KUKA KRL program: MyProgram_295().src

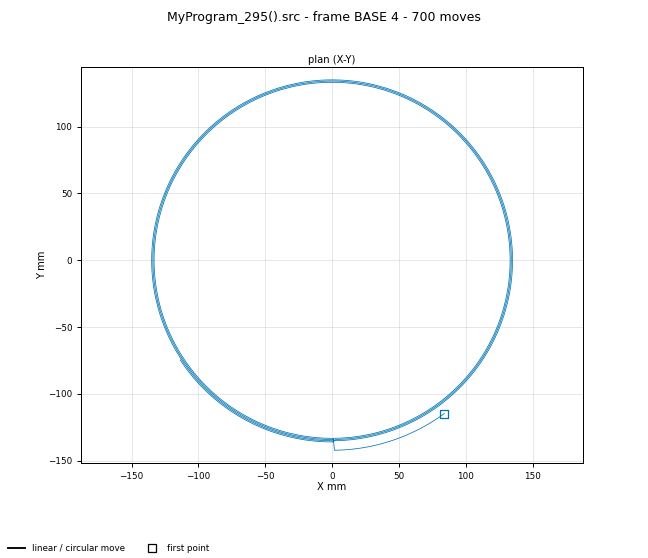
[picture p0: tool path of MyProgram_295().src in frame BASE 4, 700 of 700 moves have a stored position in this frame; points joined in program order, loops and branches not executed]
&ACCESS RVP
&REL 1
&PARAM TEMPLATE = C:\KRC\Roboter\Template\vorgabe
&PARAM EDITMASK = *
DEF MyProgram_295()
; ---- Setting reference (Base) ----
$BASE = BASE_DATA[4]

; --------------------------
; ---- Setting tool (TCP) ----
$TOOL = TOOL_DATA[3]
; --------------------------

$VEL.CP = VEL_APROX_PRINT
Startdeposition()
$VEL.CP = VEL_PRINT
LIN {X 83.9542,Y -114.6488,Z 177,A -50.7197,B 6.574,C 0.3919,E1 6.6804,E2 503.014} C_DIS
LIN {X 80.6167,Y -117.0197,Z 177,A -52.4005,B 6.5737,C 0.3953,E1 6.6765,E2 504.7003} C_DIS
LIN {X 77.4912,Y -119.1123,Z 177,A -53.839,B 6.5737,C 0.3965,E1 6.6732,E2 506.1295} C_DIS
LIN {X 74.5558,Y -120.9716,Z 177,A -55.2209,B 6.5735,C 0.3984,E1 6.6699,E2 507.51} C_DIS
LIN {X 71.534,Y -122.783,Z 177,A -56.6228,B 6.5735,C 0.4003,E1 6.6665,E2 508.9106} C_DIS
LIN {X 68.5439,Y -124.4768,Z 177,A -58.0088,B 6.5733,C 0.4024,E1 6.6632,E2 510.2978} C_DIS
LIN {X 65.0961,Y -126.3132,Z 177,A -59.6809,B 6.573,C 0.4063,E1 6.659,E2 511.9842} C_DIS
LIN {X 61.5313,Y -128.086,Z 177,A -61.1463,B 6.573,C 0.4061,E1 6.6554,E2 513.432} C_DIS
LIN {X 58.3753,Y -129.5551,Z 177,A -62.3689,B 6.5731,C 0.4049,E1 6.6523,E2 514.6314} C_DIS
LIN {X 55.9722,Y -130.6115,Z 177,A -63.5888,B 6.5729,C 0.4089,E1 6.6491,E2 515.8738} C_DIS
LIN {X 52.7667,Y -131.9389,Z 177,A -64.9738,B 6.5728,C 0.4104,E1 6.6456,E2 517.258} C_DIS
LIN {X 49.5072,Y -133.1962,Z 177,A -66.3686,B 6.5728,C 0.4117,E1 6.6419,E2 518.652} C_DIS
LIN {X 46.2416,Y -134.3648,Z 177,A -67.847,B 6.5725,C 0.4145,E1 6.638,E2 520.1421} C_DIS
LIN {X 42.8717,Y -135.4778,Z 177,A -69.1759,B 6.5725,C 0.4143,E1 6.6345,E2 521.4583} C_DIS
LIN {X 39.546,Y -136.4858,Z 177,A -70.5638,B 6.5725,C 0.4154,E1 6.6308,E2 522.8454} C_DIS
LIN {X 36.2237,Y -137.4049,Z 177,A -71.9458,B 6.5725,C 0.4164,E1 6.627,E2 524.2273} C_DIS
LIN {X 32.8538,Y -138.2496,Z 177,A -73.4276,B 6.5723,C 0.4188,E1 6.623,E2 525.7208} C_DIS
LIN {X 29.4326,Y -139.0186,Z 177,A -74.7399,B 6.5723,C 0.4182,E1 6.6194,E2 527.0204} C_DIS
LIN {X 26.0223,Y -139.6976,Z 177,A -76.1321,B 6.5723,C 0.419,E1 6.6156,E2 528.4122} C_DIS
LIN {X 22.581,Y -140.2957,Z 177,A -77.5515,B 6.5722,C 0.42,E1 6.6117,E2 529.834} C_DIS
LIN {X 19.1047,Y -140.8104,Z 177,A -78.9662,B 6.5722,C 0.4207,E1 6.6078,E2 531.2492} C_DIS
LIN {X 15.6477,Y -141.2357,Z 177,A -80.3628,B 6.5722,C 0.4212,E1 6.6039,E2 532.6455} C_DIS
LIN {X 12.1948,Y -141.5751,Z 177,A -81.8408,B 6.572,C 0.423,E1 6.5998,E2 534.1348} C_DIS
LIN {X 8.7227,Y -141.8312,Z 177,A -83.1778,B 6.572,C 0.4224,E1 6.5961,E2 535.4636} C_DIS
LIN {X 5.2085,Y -142.0041,Z 177,A -84.5529,B 6.572,C 0.4221,E1 6.5923,E2 536.8336} C_DIS
LIN {X 1.7271,Y -142.0902,Z 177,A -85.9455,B 6.572,C 0.4221,E1 6.5884,E2 538.2254} C_DIS
LIN {X 1.7271,Y -142.0902,Z 177,A -85.9455,B 6.572,C 0.4221,E1 6.5884,E2 538.2254} C_DIS
Enddeposition()
LIN {X 0.9638,Y -133.1644,Z 178,A -86.3428,B 6.5174,C 0.3854,E1 6.5313,E2 538.3182} C_DIS
Startdeposition()
$VEL.CP = VEL_PRINT
LIN {X 4.5117,Y -133.0931,Z 178,A -84.4,B 6.5178,C 0.3791,E1 6.5369,E2 536.3228} C_DIS
LIN {X 7.0319,Y -132.9825,Z 178,A -83.1818,B 6.5179,C 0.3769,E1 6.5404,E2 535.0873} C_DIS
LIN {X 10.9069,Y -132.7207,Z 178,A -81.6183,B 6.5179,C 0.3779,E1 6.5447,E2 533.5364} C_DIS
LIN {X 13.8082,Y -132.4506,Z 178,A -80.2868,B 6.5179,C 0.3763,E1 6.5484,E2 532.1945} C_DIS
LIN {X 17.4081,Y -132.025,Z 178,A -78.8233,B 6.5179,C 0.3769,E1 6.5524,E2 530.7422} C_DIS
LIN {X 21.1427,Y -131.4808,Z 178,A -77.1933,B 6.5179,C 0.3759,E1 6.5569,E2 529.1105} C_DIS
LIN {X 24.3569,Y -130.9228,Z 178,A -75.7994,B 6.518,C 0.3752,E1 6.5608,E2 527.7169} C_DIS
LIN {X 27.3232,Y -130.3367,Z 178,A -74.425,B 6.5182,C 0.3732,E1 6.5646,E2 526.3324} C_DIS
LIN {X 30.7671,Y -129.5653,Z 178,A -72.8889,B 6.5182,C 0.3718,E1 6.5687,E2 524.7932} C_DIS
LIN {X 35.009,Y -128.4853,Z 178,A -70.9984,B 6.5183,C 0.3701,E1 6.5739,E2 522.9005} C_DIS
LIN {X 39.1367,Y -127.2867,Z 178,A -69.2948,B 6.5183,C 0.3706,E1 6.5784,E2 521.2139} C_DIS
LIN {X 42.8597,Y -126.0843,Z 178,A -67.6307,B 6.5183,C 0.3692,E1 6.5828,E2 519.5511} C_DIS
LIN {X 46.8767,Y -124.6441,Z 178,A -65.7393,B 6.5185,C 0.3663,E1 6.5878,E2 517.6514} C_DIS
LIN {X 50.4594,Y -123.2392,Z 178,A -64.161,B 6.5185,C 0.3656,E1 6.5918,E2 516.0816} C_DIS
LIN {X 53.9636,Y -121.7442,Z 178,A -62.5457,B 6.5187,C 0.3639,E1 6.596,E2 514.468} C_DIS
LIN {X 56.9303,Y -120.3858,Z 178,A -61.1578,B 6.5187,C 0.3623,E1 6.5995,E2 513.0811} C_DIS
LIN {X 59.8618,Y -118.9557,Z 178,A -59.7718,B 6.5189,C 0.3606,E1 6.6029,E2 511.6962} C_DIS
LIN {X 62.7544,Y -117.4566,Z 178,A -58.3828,B 6.5189,C 0.3588,E1 6.6064,E2 510.3076} C_DIS
LIN {X 65.6366,Y -115.8708,Z 178,A -56.9757,B 6.5191,C 0.3568,E1 6.6098,E2 508.9005} C_DIS
LIN {X 68.0271,Y -114.4832,Z 178,A -55.71,B 6.5192,C 0.3538,E1 6.6129,E2 507.6242} C_DIS
LIN {X 71.6806,Y -112.2317,Z 178,A -53.8771,B 6.5194,C 0.351,E1 6.6172,E2 505.7914} C_DIS
LIN {X 74.9099,Y -110.103,Z 178,A -52.4203,B 6.5194,C 0.3515,E1 6.6205,E2 504.3592} C_DIS
LIN {X 77.5879,Y -108.2321,Z 178,A -50.9492,B 6.5195,C 0.348,E1 6.6239,E2 502.8786} C_DIS
LIN {X 80.6412,Y -105.9771,Z 178,A -49.228,B 6.5198,C 0.3437,E1 6.6278,E2 501.1451} C_DIS
LIN {X 83.8487,Y -103.4579,Z 178,A -47.5664,B 6.5198,C 0.3419,E1 6.6314,E2 499.4936} C_DIS
LIN {X 86.7837,Y -101.0083,Z 178,A -45.8978,B 6.52,C 0.3383,E1 6.635,E2 497.8205} C_DIS
LIN {X 90.026,Y -98.1295,Z 178,A -44.057,B 6.5202,C 0.335,E1 6.6388,E2 495.9812} C_DIS
LIN {X 93.0048,Y -95.3115,Z 178,A -42.3038,B 6.5204,C 0.3315,E1 6.6423,E2 494.2277} C_DIS
LIN {X 95.8799,Y -92.4185,Z 178,A -40.5795,B 6.5206,C 0.3283,E1 6.6457,E2 492.5057} C_DIS
LIN {X 98.8364,Y -89.2498,Z 178,A -38.744,B 6.5207,C 0.3247,E1 6.6491,E2 490.6721} C_DIS
LIN {X 101.7336,Y -85.9331,Z 178,A -36.8835,B 6.5209,C 0.3211,E1 6.6525,E2 488.8141} C_DIS
LIN {X 104.4775,Y -82.5752,Z 178,A -35.0437,B 6.5211,C 0.3172,E1 6.6557,E2 486.9759} C_DIS
LIN {X 106.9568,Y -79.337,Z 178,A -33.4349,B 6.5211,C 0.3156,E1 6.6584,E2 485.3836} C_DIS
LIN {X 108.8683,Y -76.6925,Z 178,A -32.0564,B 6.5213,C 0.3126,E1 6.6606,E2 484.007} C_DIS
LIN {X 111.0112,Y -73.5576,Z 178,A -30.3322,B 6.5216,C 0.3071,E1 6.6633,E2 482.2701} C_DIS
LIN {X 113.0997,Y -70.303,Z 178,A -28.7379,B 6.5217,C 0.3042,E1 6.6657,E2 480.6828} C_DIS
LIN {X 115.0507,Y -67.0639,Z 178,A -27.1021,B 6.5219,C 0.3,E1 6.668,E2 479.0444} C_DIS
LIN {X 117.2134,Y -63.207,Z 178,A -25.2998,B 6.5221,C 0.2968,E1 6.6704,E2 477.2528} C_DIS
LIN {X 118.7218,Y -60.3213,Z 178,A -23.9903,B 6.5221,C 0.2947,E1 6.6721,E2 475.9532} C_DIS
LIN {X 120.1639,Y -57.3948,Z 178,A -22.6669,B 6.5223,C 0.2924,E1 6.6737,E2 474.6386} C_DIS
LIN {X 121.5341,Y -54.4334,Z 178,A -21.1584,B 6.5225,C 0.2869,E1 6.6754,E2 473.1158} C_DIS
LIN {X 123.0296,Y -50.9648,Z 178,A -19.5935,B 6.5226,C 0.2836,E1 6.6771,E2 471.5568} C_DIS
LIN {X 124.6437,Y -46.8779,Z 178,A -17.7069,B 6.5229,C 0.2786,E1 6.679,E2 469.669} C_DIS
LIN {X 125.9218,Y -43.3284,Z 178,A -16.2072,B 6.5229,C 0.2762,E1 6.6804,E2 468.1831} C_DIS
LIN {X 126.9445,Y -40.2337,Z 178,A -14.8581,B 6.5231,C 0.2733,E1 6.6816,E2 466.8393} C_DIS
LIN {X 127.8843,Y -37.1383,Z 178,A -13.4781,B 6.5232,C 0.2696,E1 6.6827,E2 465.4595} C_DIS
LIN {X 128.7261,Y -34.1058,Z 178,A -12.1735,B 6.5234,C 0.2667,E1 6.6836,E2 464.1598} C_DIS
LIN {X 129.6834,Y -30.2687,Z 178,A -10.3349,B 6.5236,C 0.2596,E1 6.6848,E2 462.3028} C_DIS
LIN {X 130.5066,Y -26.4881,Z 178,A -8.8533,B 6.5237,C 0.258,E1 6.6857,E2 460.8423} C_DIS
LIN {X 131.1169,Y -23.281,Z 178,A -7.4791,B 6.5238,C 0.2546,E1 6.6864,E2 459.4707} C_DIS
LIN {X 131.6511,Y -20.0427,Z 178,A -6.0255,B 6.524,C 0.2499,E1 6.687,E2 458.0106} C_DIS
LIN {X 132.1671,Y -16.3023,Z 178,A -4.4968,B 6.5241,C 0.2469,E1 6.6875,E2 456.4924} C_DIS
LIN {X 132.5264,Y -13.0578,Z 178,A -3.1273,B 6.5243,C 0.2435,E1 6.6879,E2 455.126} C_DIS
LIN {X 132.8063,Y -9.8053,Z 178,A -1.7588,B 6.5243,C 0.2401,E1 6.6882,E2 453.7608} C_DIS
LIN {X 133.0068,Y -6.547,Z 178,A -0.3905,B 6.5245,C 0.2366,E1 6.6884,E2 452.3957} C_DIS
LIN {X 133.1405,Y -2.7529,Z 178,A 1.3295,B 6.5247,C 0.2305,E1 6.6886,E2 450.6637} C_DIS
LIN {X 133.1592,Y 1.6279,Z 178,A 3.1809,B 6.5249,C 0.2257,E1 6.6886,E2 448.8149} C_DIS
LIN {X 133.0343,Y 6.0011,Z 178,A 4.8481,B 6.5249,C 0.2239,E1 6.6884,E2 447.1727} C_DIS
LIN {X 132.8441,Y 9.2877,Z 178,A 6.2915,B 6.5251,C 0.2194,E1 6.6881,E2 445.7248} C_DIS
LIN {X 132.5762,Y 12.5389,Z 178,A 7.6588,B 6.5252,C 0.2161,E1 6.6878,E2 444.3609} C_DIS
LIN {X 132.2291,Y 15.7828,Z 178,A 9.0275,B 6.5253,C 0.2127,E1 6.6874,E2 442.9954} C_DIS
LIN {X 131.803,Y 19.0166,Z 178,A 10.4532,B 6.5255,C 0.2083,E1 6.6868,E2 441.566} C_DIS
LIN {X 131.2089,Y 22.7666,Z 178,A 11.9579,B 6.5255,C 0.2059,E1 6.6861,E2 440.0759} C_DIS
LIN {X 130.6108,Y 25.976,Z 178,A 13.5008,B 6.5257,C 0.1996,E1 6.6853,E2 438.5151} C_DIS
LIN {X 129.686,Y 30.2575,Z 178,A 15.1757,B 6.5257,C 0.1979,E1 6.6843,E2 436.8646} C_DIS
LIN {X 129.0503,Y 32.8574,Z 178,A 16.4149,B 6.5259,C 0.1932,E1 6.6834,E2 435.6138} C_DIS
LIN {X 128.0423,Y 36.5967,Z 178,A 17.964,B 6.526,C 0.1906,E1 6.6823,E2 434.078} C_DIS
LIN {X 127.1068,Y 39.7246,Z 178,A 19.3402,B 6.5261,C 0.1873,E1 6.6812,E2 432.7044} C_DIS
LIN {X 125.5625,Y 44.3647,Z 178,A 21.6447,B 6.5264,C 0.1782,E1 6.6791,E2 430.3742} C_DIS
LIN {X 123.8678,Y 48.8956,Z 178,A 23.4542,B 6.5264,C 0.1772,E1 6.6773,E2 428.5966} C_DIS
LIN {X 122.6601,Y 51.8494,Z 178,A 24.934,B 6.5265,C 0.1718,E1 6.6757,E2 427.1029} C_DIS
LIN {X 121.0791,Y 55.4403,Z 178,A 26.4508,B 6.5265,C 0.1703,E1 6.674,E2 425.606} C_DIS
LIN {X 119.678,Y 58.404,Z 178,A 27.8275,B 6.5266,C 0.1672,E1 6.6723,E2 424.2328} C_DIS
LIN {X 118.4793,Y 60.7976,Z 178,A 28.9716,B 6.5267,C 0.1644,E1 6.6709,E2 423.089} C_DIS
LIN {X 116.8622,Y 63.8538,Z 178,A 30.4879,B 6.5268,C 0.1602,E1 6.6688,E2 421.5685} C_DIS
LIN {X 115.0507,Y 67.0638,Z 178,A 31.9027,B 6.5268,C 0.1591,E1 6.6669,E2 420.1737} C_DIS
LIN {X 113.3731,Y 69.8617,Z 178,A 33.4559,B 6.527,C 0.1532,E1 6.6646,E2 418.6017} C_DIS
LIN {X 111.0211,Y 73.5425,Z 178,A 35.2069,B 6.527,C 0.1508,E1 6.662,E2 416.8655} C_DIS
LIN {X 109.1792,Y 76.2497,Z 178,A 36.5869,B 6.5271,C 0.148,E1 6.6598,E2 415.4883} C_DIS
LIN {X 107.2785,Y 78.9011,Z 178,A 37.925,B 6.5271,C 0.1458,E1 6.6576,E2 414.1576} C_DIS
LIN {X 105.0146,Y 81.891,Z 178,A 39.591,B 6.5273,C 0.1413,E1 6.6548,E2 412.4848} C_DIS
LIN {X 102.5253,Y 84.9859,Z 178,A 41.3184,B 6.5273,C 0.1372,E1 6.6517,E2 410.7545} C_DIS
LIN {X 99.5928,Y 88.4047,Z 178,A 43.2432,B 6.5274,C 0.1332,E1 6.6482,E2 408.8307} C_DIS
LIN {X 96.6295,Y 91.6347,Z 178,A 45.0403,B 6.5274,C 0.1307,E1 6.6448,E2 407.0439} C_DIS
LIN {X 93.806,Y 94.5224,Z 178,A 46.749,B 6.5275,C 0.1276,E1 6.6414,E2 405.3381} C_DIS
LIN {X 90.8317,Y 97.3841,Z 178,A 48.5361,B 6.5276,C 0.124,E1 6.6378,E2 403.5493} C_DIS
LIN {X 87.6175,Y 100.2858,Z 178,A 50.3796,B 6.5276,C 0.1207,E1 6.6339,E2 401.7077} C_DIS
LIN {X 84.2856,Y 103.1018,Z 178,A 52.2249,B 6.5277,C 0.1178,E1 6.63,E2 399.866} C_DIS
LIN {X 80.847,Y 105.8198,Z 178,A 54.0372,B 6.5277,C 0.1156,E1 6.626,E2 398.0623} C_DIS
LIN {X 78.3357,Y 107.6923,Z 178,A 55.396,B 6.5278,C 0.1132,E1 6.623,E2 396.702} C_DIS
LIN {X 75.4138,Y 109.758,Z 178,A 56.8258,B 6.5278,C 0.1123,E1 6.6197,E2 395.2852} C_DIS
LIN {X 72.8869,Y 111.4528,Z 178,A 58.1198,B 6.5278,C 0.1105,E1 6.6167,E2 393.993} C_DIS
LIN {X 70.3001,Y 113.1016,Z 178,A 59.529,B 6.5279,C 0.1071,E1 6.6133,E2 392.573} C_DIS
LIN {X 67.0645,Y 115.0503,Z 178,A 60.9746,B 6.5279,C 0.1074,E1 6.6099,E2 391.1489} C_DIS
LIN {X 64.6771,Y 116.4087,Z 178,A 62.2133,B 6.5279,C 0.1049,E1 6.6069,E2 389.9033} C_DIS
LIN {X 61.8012,Y 117.9582,Z 178,A 63.6121,B 6.5279,C 0.1031,E1 6.6034,E2 388.5053} C_DIS
LIN {X 58.8644,Y 119.4508,Z 178,A 65.0105,B 6.5279,C 0.1016,E1 6.5999,E2 387.1092} C_DIS
LIN {X 55.9201,Y 120.8572,Z 178,A 66.4007,B 6.528,C 0.1,E1 6.5964,E2 385.7207} C_DIS
LIN {X 52.4684,Y 122.396,Z 178,A 68.0149,B 6.528,C 0.0983,E1 6.5923,E2 384.1081} C_DIS
LIN {X 48.9807,Y 123.8348,Z 178,A 69.7866,B 6.5281,C 0.0944,E1 6.5877,E2 382.3189} C_DIS
LIN {X 44.8735,Y 125.3795,Z 178,A 71.4956,B 6.5281,C 0.0951,E1 6.5833,E2 380.6315} C_DIS
LIN {X 41.772,Y 126.4467,Z 178,A 72.8947,B 6.5281,C 0.094,E1 6.5796,E2 379.2341} C_DIS
LIN {X 38.6838,Y 127.4253,Z 178,A 74.2776,B 6.5281,C 0.093,E1 6.5759,E2 377.8527} C_DIS
LIN {X 35.5863,Y 128.3249,Z 178,A 75.6541,B 6.5281,C 0.092,E1 6.5722,E2 376.4779} C_DIS
LIN {X 32.5276,Y 129.134,Z 178,A 77.1152,B 6.5281,C 0.0896,E1 6.5682,E2 375.0052} C_DIS
LIN {X 28.0899,Y 130.1713,Z 178,A 78.9048,B 6.5281,C 0.0908,E1 6.5634,E2 373.2365} C_DIS
LIN {X 24.8792,Y 130.823,Z 178,A 80.3656,B 6.5281,C 0.0892,E1 6.5593,E2 371.77} C_DIS
LIN {X 21.6641,Y 131.3939,Z 178,A 81.7621,B 6.5281,C 0.0887,E1 6.5555,E2 370.3749} C_DIS
LIN {X 18.5251,Y 131.8732,Z 178,A 83.227,B 6.5282,C 0.0867,E1 6.5514,E2 368.8987} C_DIS
LIN {X 14.6874,Y 132.356,Z 178,A 84.7973,B 6.5282,C 0.0874,E1 6.5471,E2 367.3402} C_DIS
LIN {X 11.4395,Y 132.6757,Z 178,A 86.1979,B 6.5282,C 0.0871,E1 6.5432,E2 365.9406} C_DIS
LIN {X 8.1676,Y 132.9171,Z 178,A 87.6578,B 6.5282,C 0.0861,E1 6.5391,E2 364.4754} C_DIS
LIN {X 3.7923,Y 133.1139,Z 178,A 89.552,B 6.5282,C 0.0857,E1 6.5338,E2 362.5808} C_DIS
LIN {X 0.018,Y 133.1698,Z 178,A 91.0729,B 6.5282,C 0.0871,E1 6.5296,E2 361.073} C_DIS
LIN {X -2.7571,Y 133.1404,Z 178,A 92.4181,B 6.5282,C 0.0851,E1 6.5258,E2 359.7104} C_DIS
LIN {X -6.5309,Y 133.0076,Z 178,A 94.0135,B 6.5282,C 0.0857,E1 6.5214,E2 358.1192} C_DIS
LIN {X -10.9,Y 132.7213,Z 178,A 95.8193,B 6.5282,C 0.0871,E1 6.5164,E2 356.3236} C_DIS
LIN {X -14.16,Y 132.4128,Z 178,A 97.2257,B 6.5282,C 0.0875,E1 6.5125,E2 354.9182} C_DIS
LIN {X -17.4113,Y 132.0246,Z 178,A 98.6351,B 6.5282,C 0.0879,E1 6.5086,E2 353.5095} C_DIS
LIN {X -21.1485,Y 131.4799,Z 178,A 100.2795,B 6.5282,C 0.0884,E1 6.504,E2 351.8638} C_DIS
LIN {X -24.3644,Y 130.9214,Z 178,A 101.6857,B 6.5282,C 0.089,E1 6.5002,E2 350.4582} C_DIS
LIN {X -27.5659,Y 130.2844,Z 178,A 103.0938,B 6.5282,C 0.0898,E1 6.4963,E2 349.0505} C_DIS
LIN {X -30.7693,Y 129.5648,Z 178,A 104.6246,B 6.5282,C 0.0891,E1 6.4921,E2 347.5065} C_DIS
LIN {X -35.0164,Y 128.4833,Z 178,A 106.4004,B 6.5282,C 0.0919,E1 6.4874,E2 345.7449} C_DIS
LIN {X -37.5751,Y 127.7564,Z 178,A 107.6249,B 6.5282,C 0.0918,E1 6.484,E2 344.5116} C_DIS
LIN {X -40.7134,Y 126.7912,Z 178,A 109.0414,B 6.5282,C 0.0929,E1 6.4803,E2 343.0956} C_DIS
LIN {X -44.3614,Y 125.5637,Z 178,A 110.8869,B 6.5282,C 0.0921,E1 6.4753,E2 341.2288} C_DIS
LIN {X -48.9142,Y 123.8606,Z 178,A 112.7575,B 6.5281,C 0.097,E1 6.4705,E2 339.3859} C_DIS
LIN {X -51.9858,Y 122.6031,Z 178,A 114.3234,B 6.5281,C 0.0968,E1 6.4665,E2 337.8046} C_DIS
LIN {X -55.4531,Y 121.0732,Z 178,A 115.8357,B 6.5281,C 0.1002,E1 6.4627,E2 336.3076} C_DIS
LIN {X -58.4045,Y 119.6777,Z 178,A 117.1617,B 6.528,C 0.1028,E1 6.4593,E2 334.992} C_DIS
LIN {X -61.3202,Y 118.2108,Z 178,A 118.6541,B 6.528,C 0.1036,E1 6.4556,E2 333.4902} C_DIS
LIN {X -63.7257,Y 116.932,Z 178,A 119.9582,B 6.528,C 0.1036,E1 6.4524,E2 332.1713} C_DIS
LIN {X -66.7643,Y 115.2241,Z 178,A 121.3384,B 6.528,C 0.1071,E1 6.4491,E2 330.8065} C_DIS
LIN {X -69.4067,Y 113.6523,Z 178,A 122.82,B 6.528,C 0.1071,E1 6.4455,E2 329.3071} C_DIS
LIN {X -72.8951,Y 111.4474,Z 178,A 124.6638,B 6.5279,C 0.1091,E1 6.4411,E2 327.4566} C_DIS
LIN {X -76.1879,Y 109.2222,Z 178,A 126.2443,B 6.5279,C 0.1134,E1 6.4375,E2 325.8929} C_DIS
LIN {X -78.9118,Y 107.2706,Z 178,A 127.8007,B 6.5278,C 0.1145,E1 6.434,E2 324.324} C_DIS
LIN {X -82.3732,Y 104.6362,Z 178,A 129.6469,B 6.5278,C 0.1181,E1 6.4299,E2 322.4824} C_DIS
LIN {X -85.3094,Y 102.2571,Z 178,A 131.3251,B 6.5277,C 0.1204,E1 6.4263,E2 320.7994} C_DIS
LIN {X -88.4026,Y 99.5947,Z 178,A 133.1508,B 6.5277,C 0.1229,E1 6.4224,E2 318.9669} C_DIS
LIN {X -91.4919,Y 96.7641,Z 178,A 134.9499,B 6.5276,C 0.1265,E1 6.4188,E2 317.1698} C_DIS
LIN {X -94.5601,Y 93.7681,Z 178,A 136.7855,B 6.5275,C 0.1303,E1 6.4151,E2 315.3369} C_DIS
LIN {X -97.3895,Y 90.8259,Z 178,A 138.6197,B 6.5275,C 0.1331,E1 6.4116,E2 313.495} C_DIS
LIN {X -100.2963,Y 87.6054,Z 178,A 140.5235,B 6.5274,C 0.1366,E1 6.4081,E2 311.5884} C_DIS
LIN {X -103.1045,Y 84.2824,Z 178,A 142.4264,B 6.5273,C 0.1404,E1 6.4047,E2 309.6836} C_DIS
LIN {X -105.8227,Y 80.8432,Z 178,A 144.2965,B 6.5272,C 0.1449,E1 6.4015,E2 307.8171} C_DIS
LIN {X -107.9243,Y 78.0156,Z 178,A 145.7984,B 6.5271,C 0.1485,E1 6.399,E2 306.3182} C_DIS
LIN {X -109.811,Y 75.3366,Z 178,A 147.3294,B 6.5271,C 0.1505,E1 6.3965,E2 304.774} C_DIS
LIN {X -112.2487,Y 71.6541,Z 178,A 149.1704,B 6.5269,C 0.1558,E1 6.3937,E2 302.9418} C_DIS
LIN {X -114.2296,Y 68.4525,Z 178,A 150.8148,B 6.5269,C 0.1595,E1 6.3913,E2 301.296} C_DIS
LIN {X -115.6178,Y 66.0802,Z 178,A 152.0242,B 6.5268,C 0.1621,E1 6.3896,E2 300.0844} C_DIS
LIN {X -117.1999,Y 63.2321,Z 178,A 153.5274,B 6.5268,C 0.1645,E1 6.3876,E2 298.5704} C_DIS
LIN {X -118.7111,Y 60.3422,Z 178,A 155.0025,B 6.5266,C 0.1673,E1 6.3857,E2 297.0879} C_DIS
LIN {X -120.7967,Y 56.051,Z 178,A 157.0993,B 6.5266,C 0.1722,E1 6.3832,E2 294.9877} C_DIS
LIN {X -122.3961,Y 52.468,Z 178,A 158.7111,B 6.5264,C 0.1774,E1 6.3814,E2 293.3866} C_DIS
LIN {X -123.84,Y 48.9671,Z 178,A 160.5404,B 6.5264,C 0.1796,E1 6.3795,E2 291.5349} C_DIS
LIN {X -125.3863,Y 44.8545,Z 178,A 162.3044,B 6.5261,C 0.1861,E1 6.3778,E2 289.7877} C_DIS
LIN {X -126.4476,Y 41.769,Z 178,A 163.7384,B 6.5261,C 0.1896,E1 6.3765,E2 288.3514} C_DIS
LIN {X -127.4332,Y 38.6583,Z 178,A 165.1722,B 6.5259,C 0.1931,E1 6.3753,E2 286.9152} C_DIS
LIN {X -128.3421,Y 35.5246,Z 178,A 166.6066,B 6.5259,C 0.1967,E1 6.3743,E2 285.4785} C_DIS
LIN {X -129.1739,Y 32.3705,Z 178,A 168.1162,B 6.5257,C 0.1994,E1 6.3732,E2 283.9574} C_DIS
LIN {X -130.1662,Y 28.1131,Z 178,A 169.8859,B 6.5255,C 0.2059,E1 6.3721,E2 282.2027} C_DIS
LIN {X -130.824,Y 24.8739,Z 178,A 171.4189,B 6.5255,C 0.2087,E1 6.3713,E2 280.6576} C_DIS
LIN {X -131.3947,Y 21.6592,Z 178,A 172.8531,B 6.5253,C 0.2124,E1 6.3706,E2 279.2211} C_DIS
LIN {X -131.9575,Y 17.923,Z 178,A 174.6577,B 6.5253,C 0.2151,E1 6.3699,E2 277.3963} C_DIS
LIN {X -132.4646,Y 13.6779,Z 178,A 176.5493,B 6.5251,C 0.2198,E1 6.3693,E2 275.5} C_DIS
LIN {X -132.8073,Y 9.7921,Z 178,A 178.1203,B 6.5249,C 0.2257,E1 6.369,E2 273.9433} C_DIS
LIN {X -133.0334,Y 6.0183,Z 178,A 179.9405,B 6.5249,C 0.2283,E1 6.3687,E2 272.1011} C_DIS
LIN {X -133.159,Y 1.6377,Z 178,A -178.3452,B 6.5245,C 0.2355,E1 6.3686,E2 270.4091} C_DIS
LIN {X -133.1592,Y -1.6294,Z 178,A -176.7176,B 6.5245,C 0.2372,E1 6.3686,E2 268.7557} C_DIS
LIN {X -133.0332,Y -6.0233,Z 178,A -174.9739,B 6.5242,C 0.2442,E1 6.3688,E2 267.0314} C_DIS
LIN {X -132.8445,Y -9.2821,Z 178,A -173.4663,B 6.5242,C 0.2471,E1 6.3691,E2 265.5123} C_DIS
LIN {X -132.5763,Y -12.5379,Z 178,A -172.0358,B 6.524,C 0.2508,E1 6.3694,E2 264.0799} C_DIS
LIN {X -132.2289,Y -15.7845,Z 178,A -170.6013,B 6.5238,C 0.2545,E1 6.3699,E2 262.6428} C_DIS
LIN {X -131.8007,Y -19.0321,Z 178,A -169.1108,B 6.5238,C 0.2576,E1 6.3704,E2 261.1434} C_DIS
LIN {X -131.2089,Y -22.7668,Z 178,A -167.4875,B 6.5235,C 0.2622,E1 6.3712,E2 259.5218} C_DIS
LIN {X -130.6106,Y -25.9774,Z 178,A -166.054,B 6.5234,C 0.2658,E1 6.372,E2 258.0859} C_DIS
LIN {X -129.9358,Y -29.1637,Z 178,A -164.5219,B 6.5233,C 0.2683,E1 6.3729,E2 256.5387} C_DIS
LIN {X -128.9703,Y -33.1725,Z 178,A -162.8528,B 6.523,C 0.2744,E1 6.374,E2 254.8837} C_DIS
LIN {X -128.0384,Y -36.6106,Z 178,A -161.2582,B 6.5229,C 0.2779,E1 6.3752,E2 253.2826} C_DIS
LIN {X -127.1124,Y -39.7064,Z 178,A -159.8377,B 6.5227,C 0.2813,E1 6.3764,E2 251.8593} C_DIS
LIN {X -126.0941,Y -42.8309,Z 178,A -158.3821,B 6.5226,C 0.2847,E1 6.3776,E2 250.3995} C_DIS
LIN {X -124.6478,Y -46.8667,Z 178,A -156.4284,B 6.5224,C 0.2884,E1 6.3795,E2 248.4335} C_DIS
LIN {X -123.4191,Y -50.0133,Z 178,A -154.9576,B 6.5223,C 0.292,E1 6.3811,E2 246.9614} C_DIS
LIN {X -121.8155,Y -53.8043,Z 178,A -153.1555,B 6.5221,C 0.2963,E1 6.3831,E2 245.1565} C_DIS
LIN {X -120.3852,Y -56.9316,Z 178,A -151.8109,B 6.5218,C 0.3016,E1 6.3846,E2 243.8292} C_DIS
LIN {X -119.0565,Y -59.6637,Z 178,A -150.3536,B 6.5218,C 0.3032,E1 6.3864,E2 242.3543} C_DIS
LIN {X -117.4544,Y -62.7585,Z 178,A -148.8411,B 6.5216,C 0.3068,E1 6.3884,E2 240.8409} C_DIS
LIN {X -115.6453,Y -66.0319,Z 178,A -147.0877,B 6.5215,C 0.3091,E1 6.3908,E2 239.0705} C_DIS
LIN {X -113.3745,Y -69.8595,Z 178,A -145.1363,B 6.5213,C 0.3133,E1 6.3937,E2 237.1155} C_DIS
LIN {X -111.0145,Y -73.5526,Z 178,A -143.2028,B 6.5211,C 0.3172,E1 6.3966,E2 235.1769} C_DIS
LIN {X -108.5248,Y -77.1786,Z 178,A -141.2843,B 6.5209,C 0.3212,E1 6.3997,E2 233.2559} C_DIS
LIN {X -105.9892,Y -80.6255,Z 178,A -139.4011,B 6.5207,C 0.3249,E1 6.4028,E2 231.3683} C_DIS
LIN {X -103.4756,Y -83.8268,Z 178,A -137.6864,B 6.5205,C 0.3291,E1 6.4058,E2 229.6587} C_DIS
LIN {X -101.0063,Y -86.786,Z 178,A -135.9543,B 6.5204,C 0.3317,E1 6.409,E2 227.9179} C_DIS
LIN {X -98.1174,Y -90.0391,Z 178,A -134.0489,B 6.5202,C 0.3352,E1 6.4125,E2 226.0089} C_DIS
LIN {X -95.3144,Y -93.0018,Z 178,A -132.2472,B 6.5201,C 0.3381,E1 6.416,E2 224.2019} C_DIS
LIN {X -92.4219,Y -95.8766,Z 178,A -130.4685,B 6.5199,C 0.3412,E1 6.4196,E2 222.4206} C_DIS
LIN {X -89.4427,Y -98.6613,Z 178,A -128.699,B 6.5197,C 0.3443,E1 6.4232,E2 220.6497} C_DIS
LIN {X -86.3647,Y -101.3668,Z 178,A -126.962,B 6.5196,C 0.3478,E1 6.4269,E2 218.9162} C_DIS
LIN {X -83.2179,Y -103.9662,Z 178,A -125.1123,B 6.5195,C 0.3497,E1 6.4309,E2 217.0551} C_DIS
LIN {X -79.8155,Y -106.6005,Z 178,A -123.2351,B 6.5193,C 0.3524,E1 6.4351,E2 215.1749} C_DIS
LIN {X -76.7046,Y -108.8599,Z 178,A -121.7,B 6.5191,C 0.3565,E1 6.4386,E2 213.6548} C_DIS
LIN {X -73.5588,Y -111.0104,Z 178,A -119.8949,B 6.5191,C 0.3569,E1 6.4428,E2 211.8293} C_DIS
LIN {X -70.3041,Y -113.099,Z 178,A -118.2513,B 6.5189,C 0.3595,E1 6.4467,E2 210.1883} C_DIS
LIN {X -67.0675,Y -115.0486,Z 178,A -116.7722,B 6.5187,C 0.3636,E1 6.4502,E2 208.7274} C_DIS
LIN {X -64.8802,Y -116.2962,Z 178,A -115.6142,B 6.5187,C 0.3641,E1 6.453,E2 207.5602} C_DIS
LIN {X -61.779,Y -117.9699,Z 178,A -114.0708,B 6.5186,C 0.3656,E1 6.4568,E2 206.0132} C_DIS
LIN {X -58.8692,Y -119.4485,Z 178,A -112.6543,B 6.5185,C 0.3671,E1 6.4604,E2 204.5951} C_DIS
LIN {X -55.924,Y -120.8554,Z 178,A -111.2464,B 6.5185,C 0.3686,E1 6.4639,E2 203.1867} C_DIS
LIN {X -52.4719,Y -122.3944,Z 178,A -109.5959,B 6.5183,C 0.37,E1 6.4682,E2 201.533} C_DIS
LIN {X -48.9846,Y -123.8332,Z 178,A -107.7957,B 6.5183,C 0.3693,E1 6.4729,E2 199.7106} C_DIS
LIN {X -44.8617,Y -125.3837,Z 178,A -106.0552,B 6.5182,C 0.3729,E1 6.4774,E2 197.9891} C_DIS
LIN {X -41.7968,Y -126.4384,Z 178,A -104.6531,B 6.5182,C 0.374,E1 6.4811,E2 196.5857} C_DIS
LIN {X -38.7182,Y -127.4148,Z 178,A -103.2584,B 6.5181,C 0.3749,E1 6.4848,E2 195.1901} C_DIS
LIN {X -35.6645,Y -128.303,Z 178,A -101.8975,B 6.518,C 0.3759,E1 6.4885,E2 193.8299} C_DIS
LIN {X -32.3623,Y -129.176,Z 178,A -100.3256,B 6.518,C 0.3754,E1 6.4928,E2 192.2448} C_DIS
LIN {X -28.0815,Y -130.173,Z 178,A -98.5028,B 6.518,C 0.3773,E1 6.4977,E2 190.43} C_DIS
LIN {X -25.1996,Y -130.7617,Z 178,A -97.1703,B 6.518,C 0.377,E1 6.5014,E2 189.0888} C_DIS
LIN {X -21.6685,Y -131.3931,Z 178,A -95.6898,B 6.5179,C 0.3784,E1 6.5055,E2 187.6156} C_DIS
LIN {X -17.9346,Y -131.956,Z 178,A -94.0441,B 6.5179,C 0.3786,E1 6.51,E2 185.9667} C_DIS
LIN {X -14.6925,Y -132.3555,Z 178,A -92.6346,B 6.5179,C 0.3788,E1 6.5139,E2 184.5562} C_DIS
LIN {X -11.427,Y -132.6767,Z 178,A -91.2309,B 6.5179,C 0.3791,E1 6.5178,E2 183.1529} C_DIS
LIN {X -8.1726,Y -132.9168,Z 178,A -89.7714,B 6.5179,C 0.3784,E1 6.5219,E2 181.6859} C_DIS
LIN {X -3.8022,Y -133.1136,Z 178,A -87.8767,B 6.5179,C 0.3782,E1 6.5272,E2 179.7889} C_DIS
LIN {X -0.0979,Y -133.1694,Z 178,A -86.3929,B 6.5178,C 0.3797,E1 6.5313,E2 178.3182} C_DIS
LIN {X -0.0979,Y -133.1694,Z 178,A -86.3929,B 6.5178,C 0.3797,E1 6.5313,E2 178.3182} C_DIS
Enddeposition()
LIN {X 0.9658,Y -134.0683,Z 178,A -86.4358,B 6.517,C 0.3905,E1 6.5308,E2 178.4564} C_DIS
Startdeposition()
$VEL.CP = VEL_PRINT
LIN {X -2.4569,Y -134.0498,Z 178,A -88.0612,B 6.5169,C 0.3929,E1 6.5262,E2 180.1028} C_DIS
LIN {X -6.2008,Y -133.9296,Z 178,A -89.7044,B 6.5169,C 0.3935,E1 6.5216,E2 181.752} C_DIS
LIN {X -10.5469,Y -133.6585,Z 178,A -91.5429,B 6.5169,C 0.3931,E1 6.5165,E2 183.5885} C_DIS
LIN {X -13.8,Y -133.3609,Z 178,A -93.0256,B 6.5169,C 0.394,E1 6.5124,E2 185.0825} C_DIS
LIN {X -18.4237,Y -132.8011,Z 178,A -94.902,B 6.5169,C 0.392,E1 6.5072,E2 186.9454} C_DIS
LIN {X -22.1147,Y -132.2354,Z 178,A -96.4331,B 6.517,C 0.3905,E1 6.503,E2 188.4689} C_DIS
LIN {X -26.1073,Y -131.5069,Z 178,A -98.2587,B 6.517,C 0.3911,E1 6.498,E2 190.3064} C_DIS
LIN {X -29.6414,Y -130.7542,Z 178,A -99.7438,B 6.517,C 0.3895,E1 6.4939,E2 191.7847} C_DIS
LIN {X -33.1784,Y -129.9017,Z 178,A -101.2619,B 6.5172,C 0.3881,E1 6.4898,E2 193.2986} C_DIS
LIN {X -35.7712,Y -129.2121,Z 178,A -102.7591,B 6.5169,C 0.3921,E1 6.4857,E2 194.8397} C_DIS
LIN {X -39.0484,Y -128.2594,Z 178,A -104.5258,B 6.5168,C 0.3951,E1 6.4809,E2 196.6447} C_DIS
LIN {X -43.8026,Y -126.7144,Z 178,A -106.066,B 6.5173,C 0.3855,E1 6.477,E2 198.1116} C_DIS
LIN {X -47.9795,Y -125.1941,Z 178,A -108.0362,B 6.5173,C 0.3848,E1 6.4718,E2 200.0909} C_DIS
LIN {X -51.2597,Y -123.8863,Z 178,A -109.3526,B 6.5176,C 0.3808,E1 6.4684,E2 201.3834} C_DIS
LIN {X -54.1354,Y -122.6579,Z 178,A -110.9237,B 6.5176,C 0.3824,E1 6.4643,E2 202.9839} C_DIS
LIN {X -57.634,Y -121.0517,Z 178,A -112.4621,B 6.5176,C 0.3792,E1 6.4605,E2 204.5091} C_DIS
LIN {X -60.302,Y -119.7463,Z 178,A -113.8509,B 6.5176,C 0.3792,E1 6.457,E2 205.9128} C_DIS
LIN {X -63.9796,Y -117.8235,Z 178,A -115.6762,B 6.5178,C 0.3777,E1 6.4525,E2 207.7447} C_DIS
LIN {X -67.8599,Y -115.6319,Z 178,A -117.5757,B 6.5179,C 0.3751,E1 6.4479,E2 209.6435} C_DIS
LIN {X -71.569,Y -113.3737,Z 178,A -119.4553,B 6.5181,C 0.3728,E1 6.4434,E2 211.526} C_DIS
LIN {X -75.3391,Y -110.9043,Z 178,A -121.2915,B 6.5183,C 0.3688,E1 6.4392,E2 213.351} C_DIS
LIN {X -80.2466,Y -107.4068,Z 178,A -123.9854,B 6.5184,C 0.3662,E1 6.433,E2 216.0594} C_DIS
LIN {X -84.58,Y -104.029,Z 178,A -126.4016,B 6.5186,C 0.3631,E1 6.4277,E2 218.4836} C_DIS
LIN {X -87.9166,Y -101.2248,Z 178,A -128.3011,B 6.5188,C 0.3602,E1 6.4237,E2 220.3874} C_DIS
LIN {X -91.1167,Y -98.3543,Z 178,A -130.1213,B 6.519,C 0.3566,E1 6.4199,E2 222.2051} C_DIS
LIN {X -94.2596,Y -95.3464,Z 178,A -132.0625,B 6.5191,C 0.354,E1 6.416,E2 224.156} C_DIS
LIN {X -97.3903,Y -92.146,Z 178,A -133.9572,B 6.5193,C 0.3499,E1 6.4123,E2 226.0479} C_DIS
LIN {X -100.5171,Y -88.7245,Z 178,A -135.954,B 6.5195,C 0.3461,E1 6.4086,E2 228.0461} C_DIS
LIN {X -103.3455,Y -85.4132,Z 178,A -137.6467,B 6.5198,C 0.3401,E1 6.4056,E2 229.7174} C_DIS
LIN {X -106.0958,Y -81.9722,Z 178,A -139.7754,B 6.5199,C 0.3389,E1 6.4019,E2 231.8758} C_DIS
LIN {X -107.9322,Y -79.5385,Z 178,A -141.1068,B 6.52,C 0.3363,E1 6.3996,E2 233.2102} C_DIS
LIN {X -110.1314,Y -76.4644,Z 178,A -142.7937,B 6.5202,C 0.3334,E1 6.3969,E2 234.9052} C_DIS
LIN {X -112.7048,Y -72.6187,Z 178,A -144.8189,B 6.5204,C 0.3293,E1 6.3938,E2 236.9355} C_DIS
LIN {X -115.2608,Y -68.4887,Z 178,A -147.9219,B 6.5201,C 0.3358,E1 6.3892,E2 240.1622} C_DIS
LIN {X -118.8634,Y -62.0223,Z 178,A -150.1094,B 6.521,C 0.3171,E1 6.3865,E2 242.2298} C_DIS
LIN {X -121.3102,Y -57.0929,Z 178,A -152.4474,B 6.5213,C 0.311,E1 6.3836,E2 244.565} C_DIS
LIN {X -122.8034,Y -53.8044,Z 178,A -153.9559,B 6.5215,C 0.3066,E1 6.3819,E2 246.0684} C_DIS
LIN {X -124.1814,Y -50.5408,Z 178,A -155.5313,B 6.5216,C 0.3033,E1 6.3802,E2 247.6504} C_DIS
LIN {X -125.5343,Y -47.0779,Z 178,A -157.1382,B 6.5218,C 0.2993,E1 6.3786,E2 249.2585} C_DIS
LIN {X -126.7068,Y -43.8247,Z 178,A -158.5582,B 6.522,C 0.2948,E1 6.3773,E2 250.6706} C_DIS
LIN {X -127.7149,Y -40.7934,Z 178,A -160.1589,B 6.522,C 0.2936,E1 6.3759,E2 252.2991} C_DIS
LIN {X -128.7443,Y -37.4191,Z 178,A -161.6346,B 6.5223,C 0.2892,E1 6.3747,E2 253.77} C_DIS
LIN {X -130.0918,Y -32.4295,Z 178,A -164.2228,B 6.5223,C 0.2872,E1 6.3729,E2 256.4027} C_DIS
LIN {X -130.9048,Y -28.977,Z 178,A -165.545,B 6.5226,C 0.2809,E1 6.3721,E2 257.7005} C_DIS
LIN {X -131.6945,Y -25.1356,Z 178,A -167.1454,B 6.5229,C 0.2754,E1 6.3712,E2 259.2905} C_DIS
LIN {X -132.3941,Y -21.1539,Z 178,A -168.979,B 6.523,C 0.2717,E1 6.3703,E2 261.1357} C_DIS
LIN {X -132.9375,Y -17.4042,Z 178,A -170.5945,B 6.5232,C 0.2671,E1 6.3697,E2 262.7495} C_DIS
LIN {X -133.3978,Y -13.4432,Z 178,A -172.4256,B 6.5234,C 0.2636,E1 6.3692,E2 264.5947} C_DIS
LIN {X -133.7618,Y -9.1366,Z 178,A -174.3038,B 6.5236,C 0.2587,E1 6.3688,E2 266.4753} C_DIS
LIN {X -133.9946,Y -4.6002,Z 178,A -176.3053,B 6.5238,C 0.2538,E1 6.3685,E2 268.4826} C_DIS
LIN {X -134.0725,Y -0.3422,Z 178,A -178.1529,B 6.5239,C 0.2488,E1 6.3685,E2 270.332} C_DIS
LIN {X -134.0188,Y 3.7792,Z 178,A -179.8716,B 6.5242,C 0.2433,E1 6.3685,E2 272.044} C_DIS
LIN {X -133.8444,Y 7.8207,Z 178,A 178.3411,B 6.5243,C 0.239,E1 6.3688,E2 273.837} C_DIS
LIN {X -133.5759,Y 11.5256,Z 178,A 176.6892,B 6.5244,C 0.2352,E1 6.3692,E2 275.4954} C_DIS
LIN {X -133.1951,Y 15.3191,Z 178,A 174.9893,B 6.5246,C 0.2313,E1 6.3697,E2 277.2023} C_DIS
LIN {X -132.7202,Y 18.9902,Z 178,A 173.4768,B 6.5248,C 0.226,E1 6.3703,E2 278.7051} C_DIS
LIN {X -132.1442,Y 22.6613,Z 178,A 171.8771,B 6.5249,C 0.2217,E1 6.371,E2 280.3048} C_DIS
LIN {X -131.4626,Y 26.3251,Z 178,A 170.1889,B 6.525,C 0.2182,E1 6.3719,E2 282.0031} C_DIS
LIN {X -130.7231,Y 29.7775,Z 178,A 168.5673,B 6.5251,C 0.2152,E1 6.3729,E2 283.6369} C_DIS
LIN {X -129.7115,Y 33.9198,Z 178,A 166.7486,B 6.5253,C 0.21,E1 6.3741,E2 285.4536} C_DIS
LIN {X -128.8931,Y 36.911,Z 178,A 165.4895,B 6.5254,C 0.2057,E1 6.3751,E2 286.7036} C_DIS
LIN {X -127.8549,Y 40.3551,Z 178,A 164.0474,B 6.5256,C 0.2004,E1 6.3762,E2 288.1329} C_DIS
LIN {X -126.73,Y 43.7576,Z 178,A 162.505,B 6.5257,C 0.1964,E1 6.3776,E2 289.6751} C_DIS
LIN {X -125.5126,Y 47.1359,Z 178,A 160.7304,B 6.5257,C 0.1948,E1 6.3793,E2 291.4771} C_DIS
LIN {X -123.9387,Y 51.1342,Z 178,A 158.8278,B 6.5259,C 0.1906,E1 6.3813,E2 293.386} C_DIS
LIN {X -122.5902,Y 54.2868,Z 178,A 157.1909,B 6.5259,C 0.1886,E1 6.3832,E2 295.0421} C_DIS
LIN {X -120.4809,Y 58.8202,Z 178,A 155.0303,B 6.5261,C 0.1833,E1 6.3858,E2 297.2036} C_DIS
LIN {X -118.329,Y 63.04,Z 178,A 153.0296,B 6.5263,C 0.1779,E1 6.3883,E2 299.1996} C_DIS
LIN {X -116.3225,Y 66.6697,Z 178,A 151.2335,B 6.5263,C 0.1738,E1 6.3908,E2 300.9968} C_DIS
LIN {X -114.14,Y 70.3409,Z 178,A 149.4893,B 6.5265,C 0.1684,E1 6.3933,E2 302.7298} C_DIS
LIN {X -110.8859,Y 75.3663,Z 178,A 146.7819,B 6.5266,C 0.1639,E1 6.3975,E2 305.4525} C_DIS
LIN {X -108.3784,Y 78.9299,Z 178,A 144.9508,B 6.5267,C 0.1592,E1 6.4004,E2 307.2783} C_DIS
LIN {X -105.8629,Y 82.2726,Z 178,A 143.0538,B 6.5268,C 0.1563,E1 6.4037,E2 309.1867} C_DIS
LIN {X -103.0477,Y 85.7729,Z 178,A 141.0836,B 6.5268,C 0.1526,E1 6.4072,E2 311.161} C_DIS
LIN {X -100.1457,Y 89.1443,Z 178,A 139.1423,B 6.527,C 0.149,E1 6.4107,E2 313.1055} C_DIS
LIN {X -97.333,Y 92.2066,Z 178,A 137.3837,B 6.527,C 0.145,E1 6.4141,E2 314.8603} C_DIS
LIN {X -94.333,Y 95.2735,Z 178,A 135.4778,B 6.5271,C 0.1421,E1 6.4179,E2 316.7731} C_DIS
LIN {X -91.1407,Y 98.3319,Z 178,A 133.5661,B 6.5272,C 0.1387,E1 6.4217,E2 318.6859} C_DIS
LIN {X -87.894,Y 101.2446,Z 178,A 131.6636,B 6.5272,C 0.1356,E1 6.4257,E2 320.5914} C_DIS
LIN {X -84.5164,Y 104.081,Z 178,A 129.763,B 6.5273,C 0.1323,E1 6.4298,E2 322.4922} C_DIS
LIN {X -81.0572,Y 106.7969,Z 178,A 127.8299,B 6.5273,C 0.1297,E1 6.4341,E2 324.43} C_DIS
LIN {X -76.9535,Y 109.7908,Z 178,A 125.239,B 6.5273,C 0.131,E1 6.4401,E2 327.0686} C_DIS
LIN {X -73.3141,Y 112.2536,Z 178,A 123.6334,B 6.5275,C 0.1248,E1 6.4438,E2 328.6407} C_DIS
LIN {X -69.2276,Y 114.8185,Z 178,A 121.6664,B 6.5275,C 0.1206,E1 6.4484,E2 330.5948} C_DIS
LIN {X -65.7694,Y 116.8336,Z 178,A 119.5762,B 6.5275,C 0.1228,E1 6.4536,E2 332.7284} C_DIS
LIN {X -62.2721,Y 118.7322,Z 178,A 118.2756,B 6.5276,C 0.1157,E1 6.4567,E2 333.9805} C_DIS
LIN {X -58.5289,Y 120.6242,Z 178,A 116.4274,B 6.5276,C 0.1141,E1 6.4613,E2 335.8341} C_DIS
LIN {X -55.5007,Y 122.0472,Z 178,A 115.0525,B 6.5277,C 0.1118,E1 6.4648,E2 337.2014} C_DIS
LIN {X -51.7704,Y 123.673,Z 178,A 113.3461,B 6.5277,C 0.1094,E1 6.4692,E2 338.9025} C_DIS
LIN {X -44.5398,Y 126.4588,Z 178,A 109.8829,B 6.5277,C 0.108,E1 6.4783,E2 342.3816} C_DIS
LIN {X -41.0724,Y 127.6258,Z 178,A 107.903,B 6.5277,C 0.1118,E1 6.4837,E2 344.4093} C_DIS
LIN {X -36.8436,Y 128.9122,Z 178,A 106.3458,B 6.5278,C 0.1062,E1 6.4877,E2 345.9265} C_DIS
LIN {X -33.1154,Y 129.9177,Z 178,A 104.8228,B 6.5278,C 0.1034,E1 6.4918,E2 347.4333} C_DIS
LIN {X -29.7248,Y 130.7352,Z 178,A 103.3403,B 6.5278,C 0.1023,E1 6.4958,E2 348.9139} C_DIS
LIN {X -25.8764,Y 131.5529,Z 178,A 101.5378,B 6.5278,C 0.103,E1 6.5008,E2 350.7298} C_DIS
LIN {X -21.7794,Y 132.2913,Z 178,A 99.7719,B 6.5278,C 0.102,E1 6.5056,E2 352.4931} C_DIS
LIN {X -17.6089,Y 132.9106,Z 178,A 98.0824,B 6.5279,C 0.0998,E1 6.5103,E2 354.1683} C_DIS
LIN {X -14.6697,Y 133.2674,Z 178,A 96.9064,B 6.5279,C 0.0982,E1 6.5135,E2 355.333} C_DIS
LIN {X -12.2933,Y 133.5082,Z 178,A 95.7991,B 6.5279,C 0.0991,E1 6.5166,E2 356.4502} C_DIS
LIN {X -8.5752,Y 133.7979,Z 178,A 94.2924,B 6.5279,C 0.0976,E1 6.5208,E2 357.9457} C_DIS
LIN {X -5.6239,Y 133.9546,Z 178,A 92.8152,B 6.5279,C 0.1004,E1 6.525,E2 359.4476} C_DIS
LIN {X -2.1679,Y 134.0546,Z 178,A 91.4698,B 6.5279,C 0.0985,E1 6.5287,E2 360.7767} C_DIS
LIN {X 1.354,Y 134.0667,Z 178,A 89.8351,B 6.5279,C 0.1003,E1 6.5333,E2 362.4261} C_DIS
LIN {X 5.0613,Y 133.9766,Z 178,A 88.3336,B 6.5279,C 0.0994,E1 6.5375,E2 363.9171} C_DIS
LIN {X 8.4946,Y 133.8029,Z 178,A 86.8158,B 6.5279,C 0.1003,E1 6.5417,E2 365.44} C_DIS
LIN {X 13.7764,Y 133.3635,Z 178,A 84.5349,B 6.5279,C 0.1011,E1 6.5481,E2 367.722} C_DIS
LIN {X 17.7577,Y 132.8911,Z 178,A 82.8484,B 6.5279,C 0.1014,E1 6.5527,E2 369.4048} C_DIS
LIN {X 22.0616,Y 132.2443,Z 178,A 81.1448,B 6.5279,C 0.1001,E1 6.5574,E2 371.0892} C_DIS
LIN {X 24.9533,Y 131.7294,Z 178,A 79.8384,B 6.5279,C 0.1014,E1 6.561,E2 372.4013} C_DIS
LIN {X 28.3342,Y 131.0436,Z 178,A 78.3409,B 6.5279,C 0.1027,E1 6.5651,E2 373.9012} C_DIS
LIN {X 32.2695,Y 130.1324,Z 178,A 76.1974,B 6.5277,C 0.1098,E1 6.571,E2 376.0937} C_DIS
LIN {X 35.9456,Y 129.1633,Z 178,A 74.3936,B 6.5277,C 0.1136,E1 6.5759,E2 377.9182} C_DIS
LIN {X 40.6689,Y 127.7547,Z 178,A 72.8615,B 6.5277,C 0.1072,E1 6.5798,E2 379.3821} C_DIS
LIN {X 45.6635,Y 126.0559,Z 178,A 70.6503,B 6.5277,C 0.1087,E1 6.5857,E2 381.5878} C_DIS
LIN {X 49.5486,Y 124.5813,Z 178,A 68.8272,B 6.5277,C 0.1113,E1 6.5904,E2 383.4163} C_DIS
LIN {X 53.0324,Y 123.1372,Z 178,A 67.2992,B 6.5277,C 0.1118,E1 6.5943,E2 384.9341} C_DIS
LIN {X 56.1163,Y 121.7627,Z 178,A 65.9871,B 6.5277,C 0.1116,E1 6.5976,E2 386.2305} C_DIS
LIN {X 58.9039,Y 120.4396,Z 178,A 64.5227,B 6.5277,C 0.1154,E1 6.6013,E2 387.7123} C_DIS
LIN {X 62.2156,Y 118.7619,Z 178,A 63.0498,B 6.5277,C 0.1158,E1 6.605,E2 389.1715} C_DIS
LIN {X 65.4624,Y 117.0062,Z 178,A 61.3312,B 6.5276,C 0.1201,E1 6.6092,E2 390.907} C_DIS
LIN {X 69.47,Y 114.6719,Z 178,A 59.4498,B 6.5276,C 0.1215,E1 6.6137,E2 392.7765} C_DIS
LIN {X 73.0172,Y 112.4464,Z 178,A 57.0788,B 6.5273,C 0.1332,E1 6.6194,E2 395.2166} C_DIS
LIN {X 77.2598,Y 109.5747,Z 178,A 55.4682,B 6.5274,C 0.1279,E1 6.623,E2 396.7588} C_DIS
LIN {X 80.8613,Y 106.9447,Z 178,A 53.6116,B 6.5274,C 0.1304,E1 6.6271,E2 398.6097} C_DIS
LIN {X 84.4048,Y 104.1711,Z 178,A 51.6879,B 6.5274,C 0.1338,E1 6.6313,E2 400.5338} C_DIS
LIN {X 87.755,Y 101.3651,Z 178,A 50.1057,B 6.5274,C 0.1328,E1 6.6346,E2 402.0822} C_DIS
LIN {X 90.4494,Y 98.9685,Z 178,A 48.3158,B 6.5272,C 0.1397,E1 6.6384,E2 403.9022} C_DIS
LIN {X 93.5167,Y 96.0752,Z 178,A 46.5463,B 6.5272,C 0.1428,E1 6.642,E2 405.6683} C_DIS
LIN {X 95.9688,Y 93.6259,Z 178,A 45.059,B 6.527,C 0.1459,E1 6.6449,E2 407.1567} C_DIS
LIN {X 99.0635,Y 90.3451,Z 178,A 43.1998,B 6.527,C 0.1488,E1 6.6484,E2 409.0083} C_DIS
LIN {X 101.9573,Y 87.0661,Z 178,A 40.5046,B 6.5266,C 0.1661,E1 6.6535,E2 411.8025} C_DIS
LIN {X 106.2313,Y 81.7963,Z 178,A 38.4827,B 6.5268,C 0.1585,E1 6.6568,E2 413.7209} C_DIS
LIN {X 108.9146,Y 78.188,Z 178,A 36.6089,B 6.5267,C 0.1622,E1 6.6598,E2 415.5896} C_DIS
LIN {X 111.3304,Y 74.7084,Z 178,A 34.8704,B 6.5266,C 0.1653,E1 6.6626,E2 417.3203} C_DIS
LIN {X 113.6702,Y 71.0978,Z 178,A 33.038,B 6.5265,C 0.1696,E1 6.6653,E2 419.1528} C_DIS
LIN {X 115.9833,Y 67.2576,Z 178,A 31.1718,B 6.5264,C 0.1735,E1 6.668,E2 421.0138} C_DIS
LIN {X 118.1653,Y 63.3457,Z 178,A 29.2817,B 6.5263,C 0.1779,E1 6.6705,E2 422.902} C_DIS
LIN {X 120.0738,Y 59.6454,Z 178,A 27.6392,B 6.5262,C 0.1802,E1 6.6726,E2 424.5288} C_DIS
LIN {X 121.4952,Y 56.6948,Z 178,A 26.3797,B 6.5262,C 0.1815,E1 6.6741,E2 425.7721} C_DIS
LIN {X 123.1372,Y 53.0324,Z 178,A 24.2867,B 6.5258,C 0.1922,E1 6.6765,E2 427.9116} C_DIS
LIN {X 124.4031,Y 49.9906,Z 178,A 22.3422,B 6.5255,C 0.2048,E1 6.6785,E2 429.9214} C_DIS
LIN {X 126.624,Y 44.0633,Z 178,A 20.8142,B 6.5258,C 0.1925,E1 6.6798,E2 431.309} C_DIS
LIN {X 127.9674,Y 40.0024,Z 178,A 18.7688,B 6.5256,C 0.2011,E1 6.6816,E2 433.3822} C_DIS
LIN {X 128.9091,Y 36.8547,Z 178,A 17.3486,B 6.5255,C 0.2053,E1 6.6827,E2 434.8053} C_DIS
LIN {X 129.8589,Y 33.347,Z 178,A 15.8485,B 6.5253,C 0.2087,E1 6.6838,E2 436.2999} C_DIS
LIN {X 130.6659,Y 30.0281,Z 178,A 14.4449,B 6.5253,C 0.2118,E1 6.6847,E2 437.6976} C_DIS
LIN {X 131.3345,Y 26.9544,Z 178,A 13.2052,B 6.5252,C 0.2138,E1 6.6854,E2 438.9255} C_DIS
LIN {X 131.9373,Y 23.8296,Z 178,A 11.7806,B 6.525,C 0.2187,E1 6.6862,E2 440.359} C_DIS
LIN {X 132.6036,Y 19.8004,Z 178,A 9.992,B 6.5248,C 0.2243,E1 6.6869,E2 442.1542} C_DIS
LIN {X 133.0955,Y 16.1536,Z 178,A 8.6641,B 6.5248,C 0.2246,E1 6.6874,E2 443.4534} C_DIS
LIN {X 133.3804,Y 13.6192,Z 178,A 7.3543,B 6.5246,C 0.2315,E1 6.6878,E2 444.7909} C_DIS
LIN {X 133.7158,Y 9.7665,Z 178,A 5.8624,B 6.5246,C 0.2335,E1 6.6881,E2 446.2644} C_DIS
LIN {X 133.9133,Y 6.5257,Z 178,A 4.3924,B 6.5243,C 0.2388,E1 6.6883,E2 447.7456} C_DIS
LIN {X 134.063,Y 1.66,Z 178,A 2.3809,B 6.5241,C 0.2436,E1 6.6885,E2 449.7504} C_DIS
LIN {X 134.0472,Y -2.6133,Z 178,A 0.7124,B 6.5241,C 0.2462,E1 6.6885,E2 451.4011} C_DIS
LIN {X 133.9577,Y -5.5463,Z 178,A -0.8365,B 6.5237,C 0.2548,E1 6.6883,E2 452.987} C_DIS
LIN {X 133.7734,Y -8.9723,Z 178,A -2.1399,B 6.5237,C 0.2562,E1 6.688,E2 454.2719} C_DIS
LIN {X 133.4111,Y -13.3045,Z 178,A -3.8229,B 6.5236,C 0.2586,E1 6.6876,E2 455.9349} C_DIS
LIN {X 132.9513,Y -17.2988,Z 178,A -5.5518,B 6.5234,C 0.2636,E1 6.687,E2 457.6667} C_DIS
LIN {X 132.3169,Y -21.6265,Z 178,A -7.491,B 6.5231,C 0.2701,E1 6.6862,E2 459.616} C_DIS
LIN {X 131.4001,Y -26.6319,Z 178,A -9.4476,B 6.523,C 0.2726,E1 6.6852,E2 461.5478} C_DIS
LIN {X 130.6802,Y -29.9654,Z 178,A -10.782,B 6.523,C 0.2746,E1 6.6844,E2 462.8683} C_DIS
LIN {X 128.8323,Y -37.1184,Z 178,A -14.0709,B 6.5224,C 0.2857,E1 6.682,E2 466.1764} C_DIS
LIN {X 127.7646,Y -40.638,Z 178,A -15.6191,B 6.5223,C 0.2896,E1 6.6807,E2 467.7231} C_DIS
LIN {X 126.3287,Y -44.9066,Z 178,A -17.4339,B 6.5221,C 0.293,E1 6.6791,E2 469.5262} C_DIS
LIN {X 125.3253,Y -47.6359,Z 178,A -18.6379,B 6.522,C 0.2957,E1 6.6779,E2 470.7265} C_DIS
LIN {X 123.8205,Y -51.4171,Z 178,A -20.2916,B 6.5219,C 0.2989,E1 6.6762,E2 472.3712} C_DIS
LIN {X 122.4105,Y -54.6887,Z 178,A -21.7176,B 6.5217,C 0.3013,E1 6.6746,E2 473.7868} C_DIS
LIN {X 121.3284,Y -57.0545,Z 178,A -23.0316,B 6.5214,C 0.3077,E1 6.673,E2 475.1269} C_DIS
LIN {X 119.6559,Y -60.4795,Z 178,A -24.4929,B 6.5214,C 0.3091,E1 6.6712,E2 476.569} C_DIS
LIN {X 117.0855,Y -65.3212,Z 178,A -26.8554,B 6.5211,C 0.3154,E1 6.668,E2 478.9362} C_DIS
LIN {X 114.9472,Y -69.0147,Z 178,A -28.6404,B 6.5209,C 0.3194,E1 6.6655,E2 480.718} C_DIS
LIN {X 112.8351,Y -72.4152,Z 178,A -30.2645,B 6.5208,C 0.3221,E1 6.6631,E2 482.333} C_DIS
LIN {X 110.4048,Y -76.0693,Z 178,A -32.16,B 6.5205,C 0.327,E1 6.6601,E2 484.2328} C_DIS
LIN {X 107.8255,Y -79.6839,Z 178,A -34.0449,B 6.5203,C 0.3313,E1 6.657,E2 486.1179} C_DIS
LIN {X 105.1045,Y -83.2398,Z 178,A -35.9339,B 6.5201,C 0.3353,E1 6.6538,E2 488.0056} C_DIS
LIN {X 102.1347,Y -86.8574,Z 178,A -37.8032,B 6.52,C 0.3377,E1 6.6505,E2 489.8604} C_DIS
LIN {X 99.5654,Y -89.792,Z 178,A -39.5413,B 6.5197,C 0.3425,E1 6.6472,E2 491.609} C_DIS
LIN {X 96.6587,Y -92.9137,Z 178,A -41.3033,B 6.5196,C 0.3455,E1 6.6439,E2 493.3651} C_DIS
LIN {X 93.768,Y -95.8295,Z 178,A -42.7981,B 6.5196,C 0.3449,E1 6.641,E2 494.8291} C_DIS
LIN {X 90.7713,Y -98.6726,Z 178,A -44.7658,B 6.5192,C 0.3518,E1 6.6369,E2 496.8237} C_DIS
LIN {X 87.4287,Y -101.6461,Z 178,A -46.5855,B 6.5192,C 0.354,E1 6.6331,E2 498.6336} C_DIS
LIN {X 84.4225,Y -104.1569,Z 178,A -48.3314,B 6.5189,C 0.3584,E1 6.6293,E2 500.39} C_DIS
LIN {X 80.8274,Y -106.9703,Z 178,A -50.2007,B 6.5187,C 0.3607,E1 6.6252,E2 502.2508} C_DIS
LIN {X 77.5799,Y -109.349,Z 178,A -51.9526,B 6.5185,C 0.3642,E1 6.6212,E2 504.008} C_DIS
LIN {X 74.049,Y -111.7703,Z 178,A -53.7607,B 6.5184,C 0.3669,E1 6.617,E2 505.8151} C_DIS
LIN {X 70.4569,Y -114.0688,Z 178,A -55.5608,B 6.5182,C 0.3695,E1 6.6128,E2 507.6138} C_DIS
LIN {X 66.5415,Y -116.3956,Z 178,A -57.4252,B 6.5182,C 0.3712,E1 6.6083,E2 509.4696} C_DIS
LIN {X 62.9886,Y -118.356,Z 178,A -59.1746,B 6.518,C 0.374,E1 6.604,E2 511.2223} C_DIS
LIN {X 59.5706,Y -120.1107,Z 178,A -60.5046,B 6.5181,C 0.3714,E1 6.6008,E2 512.5145} C_DIS
LIN {X 56.3291,Y -121.6643,Z 178,A -62.0829,B 6.518,C 0.3741,E1 6.5968,E2 514.0993} C_DIS
LIN {X 54.0741,Y -122.6854,Z 178,A -63.2516,B 6.5178,C 0.3772,E1 6.5938,E2 515.2827} C_DIS
LIN {X 48.6645,Y -124.9278,Z 178,A -65.6938,B 6.5177,C 0.3792,E1 6.5875,E2 517.7193} C_DIS
LIN {X 45.9433,Y -125.955,Z 178,A -66.8381,B 6.5177,C 0.3792,E1 6.5845,E2 518.8522} C_DIS
LIN {X 40.8774,Y -127.6881,Z 178,A -69.219,B 6.5175,C 0.3829,E1 6.5782,E2 521.2463} C_DIS
LIN {X 37.8401,Y -128.621,Z 178,A -70.5587,B 6.5175,C 0.3839,E1 6.5746,E2 522.5847} C_DIS
LIN {X 34.4967,Y -129.5577,Z 178,A -72.1333,B 6.5173,C 0.3865,E1 6.5703,E2 524.1716} C_DIS
LIN {X 30.1559,Y -130.6367,Z 178,A -73.8229,B 6.5173,C 0.3847,E1 6.5658,E2 525.8347} C_DIS
LIN {X 26.9177,Y -131.342,Z 178,A -75.3015,B 6.5173,C 0.3867,E1 6.5617,E2 527.322} C_DIS
LIN {X 22.7523,Y -132.129,Z 178,A -77.219,B 6.5171,C 0.3894,E1 6.5564,E2 529.2539} C_DIS
LIN {X 19.7925,Y -132.6049,Z 178,A -78.4221,B 6.5171,C 0.3889,E1 6.5531,E2 530.448} C_DIS
LIN {X 16.1491,Y -133.096,Z 178,A -80.0578,B 6.5171,C 0.3907,E1 6.5486,E2 532.0927} C_DIS
LIN {X 11.3889,Y -133.5874,Z 178,A -81.9186,B 6.5171,C 0.3888,E1 6.5435,E2 533.9315} C_DIS
LIN {X 6.115,Y -133.9339,Z 178,A -84.2676,B 6.5171,C 0.3908,E1 6.5369,E2 536.2931} C_DIS
LIN {X 2.6729,Y -134.0462,Z 178,A -85.7507,B 6.517,C 0.3912,E1 6.5327,E2 537.7783} C_DIS
LIN {X 2.6729,Y -134.0462,Z 178,A -85.7507,B 6.517,C 0.3912,E1 6.5327,E2 537.7783} C_DIS
Enddeposition()
LIN {X 0.9756,Y -134.971,Z 178,A -85.9682,B 6.5172,C 0.3877,E1 6.5322,E2 537.9649} C_DIS
Startdeposition()
$VEL.CP = VEL_PRINT
LIN {X 4.5844,Y -134.9001,Z 178,A -83.8164,B 6.5177,C 0.3783,E1 6.5384,E2 535.7333} C_DIS
LIN {X 8.8066,Y -134.6896,Z 178,A -82.5459,B 6.5173,C 0.3856,E1 6.5418,E2 534.529} C_DIS
LIN {X 14.316,Y -134.2149,Z 178,A -80.4411,B 6.5171,C 0.3883,E1 6.5476,E2 532.4538} C_DIS
LIN {X 17.4026,Y -133.8496,Z 178,A -78.8238,B 6.5174,C 0.3832,E1 6.5521,E2 530.7978} C_DIS
LIN {X 21.458,Y -133.2617,Z 178,A -76.8423,B 6.5177,C 0.3786,E1 6.5577,E2 528.7844} C_DIS
LIN {X 25.9081,Y -132.4675,Z 178,A -75.1676,B 6.5176,C 0.3811,E1 6.5622,E2 527.1397} C_DIS
LIN {X 29.8295,Y -131.6388,Z 178,A -73.507,B 6.5176,C 0.3804,E1 6.5667,E2 525.4833} C_DIS
LIN {X 33.2829,Y -130.8081,Z 178,A -72.0083,B 6.5176,C 0.3794,E1 6.5708,E2 523.9847} C_DIS
LIN {X 37.0364,Y -129.7972,Z 178,A -70.4082,B 6.5176,C 0.3787,E1 6.5751,E2 522.39} C_DIS
LIN {X 39.5453,Y -129.0529,Z 178,A -69.2694,B 6.5178,C 0.3772,E1 6.5781,E2 521.2467} C_DIS
LIN {X 44.3662,Y -127.476,Z 178,A -67.0991,B 6.5179,C 0.3747,E1 6.5839,E2 519.0728} C_DIS
LIN {X 48.1076,Y -126.1132,Z 178,A -64.765,B 6.5186,C 0.3627,E1 6.5902,E2 516.6548} C_DIS
LIN {X 53.1499,Y -124.0715,Z 178,A -63.3293,B 6.518,C 0.3737,E1 6.5936,E2 515.3294} C_DIS
LIN {X 55.7318,Y -122.9345,Z 178,A -61.9996,B 6.5182,C 0.3701,E1 6.5971,E2 513.982} C_DIS
LIN {X 59.1782,Y -121.3126,Z 178,A -60.1289,B 6.5185,C 0.3639,E1 6.6019,E2 512.0775} C_DIS
LIN {X 62.0516,Y -119.8693,Z 178,A -59.0681,B 6.5184,C 0.3668,E1 6.6044,E2 511.0545} C_DIS
LIN {X 65.0444,Y -118.2724,Z 178,A -57.4919,B 6.5186,C 0.3625,E1 6.6083,E2 509.4599} C_DIS
LIN {X 68.8682,Y -116.0872,Z 178,A -55.6508,B 6.5187,C 0.3601,E1 6.6127,E2 507.6209} C_DIS
LIN {X 72.8629,Y -113.6222,Z 178,A -53.719,B 6.5189,C 0.3579,E1 6.6173,E2 505.6951} C_DIS
LIN {X 76.6288,Y -111.1175,Z 178,A -51.8036,B 6.519,C 0.3547,E1 6.6217,E2 503.7787} C_DIS
LIN {X 80.0203,Y -108.7003,Z 178,A -50.093,B 6.5192,C 0.3525,E1 6.6256,E2 502.0738} C_DIS
LIN {X 83.5415,Y -106.0182,Z 178,A -48.2484,B 6.5193,C 0.3496,E1 6.6296,E2 500.232} C_DIS
LIN {X 86.7855,Y -103.3792,Z 178,A -46.4879,B 6.5195,C 0.3465,E1 6.6334,E2 498.4718} C_DIS
LIN {X 90.1229,Y -100.4831,Z 178,A -44.0215,B 6.5202,C 0.3329,E1 6.6387,E2 495.9281} C_DIS
LIN {X 94.1329,Y -96.7373,Z 178,A -42.6072,B 6.5196,C 0.3434,E1 6.6414,E2 494.6287} C_DIS
LIN {X 97.4329,Y -93.4123,Z 178,A -40.3615,B 6.5201,C 0.3349,E1 6.6458,E2 492.3485} C_DIS
LIN {X 100.4818,Y -90.1244,Z 178,A -38.5694,B 6.5201,C 0.3326,E1 6.6492,E2 490.5687} C_DIS
LIN {X 103.1313,Y -87.081,Z 178,A -36.7807,B 6.5205,C 0.3275,E1 6.6524,E2 488.7688} C_DIS
LIN {X 106.0161,Y -83.5441,Z 178,A -34.9256,B 6.5206,C 0.3244,E1 6.6557,E2 486.9224} C_DIS
LIN {X 108.6649,Y -80.0685,Z 178,A -33.0951,B 6.5208,C 0.3205,E1 6.6587,E2 485.0933} C_DIS
LIN {X 111.204,Y -76.5028,Z 178,A -31.2596,B 6.521,C 0.3164,E1 6.6617,E2 483.259} C_DIS
LIN {X 113.7849,Y -72.6087,Z 178,A -29.359,B 6.5212,C 0.313,E1 6.6645,E2 481.3669} C_DIS
LIN {X 116.0295,Y -68.9649,Z 178,A -27.5541,B 6.5214,C 0.3086,E1 6.6671,E2 479.5618} C_DIS
LIN {X 118.1659,Y -65.2367,Z 178,A -25.2143,B 6.522,C 0.2951,E1 6.6704,E2 477.1547} C_DIS
LIN {X 120.5403,Y -60.7354,Z 178,A -23.769,B 6.5217,C 0.3018,E1 6.6721,E2 475.7982} C_DIS
LIN {X 121.8711,Y -58.0165,Z 178,A -22.4486,B 6.5219,C 0.2979,E1 6.6737,E2 474.4721} C_DIS
LIN {X 123.2868,Y -54.944,Z 178,A -21.0452,B 6.522,C 0.2946,E1 6.6754,E2 473.0714} C_DIS
LIN {X 124.9484,Y -51.0566,Z 178,A -18.8683,B 6.5225,C 0.2832,E1 6.6777,E2 470.8444} C_DIS
LIN {X 126.3976,Y -47.3509,Z 178,A -17.6864,B 6.5223,C 0.2874,E1 6.6788,E2 469.7252} C_DIS
LIN {X 128.2852,Y -41.9747,Z 178,A -15.3084,B 6.5226,C 0.2815,E1 6.681,E2 467.3502} C_DIS
LIN {X 129.1792,Y -39.1328,Z 178,A -14.0561,B 6.5227,C 0.2782,E1 6.682,E2 466.0983} C_DIS
LIN {X 130.7286,Y -33.5949,Z 178,A -11.614,B 6.523,C 0.2714,E1 6.6838,E2 463.6538} C_DIS
LIN {X 131.5762,Y -30.1036,Z 178,A -10.1429,B 6.5232,C 0.2681,E1 6.6848,E2 462.1881} C_DIS
LIN {X 132.3596,Y -26.4516,Z 178,A -8.6185,B 6.5232,C 0.2647,E1 6.6856,E2 460.6701} C_DIS
LIN {X 133.2013,Y -21.8199,Z 178,A -6.622,B 6.5235,C 0.259,E1 6.6866,E2 458.672} C_DIS
LIN {X 133.7956,Y -17.8145,Z 178,A -4.9548,B 6.5237,C 0.255,E1 6.6872,E2 457.0098} C_DIS
LIN {X 134.2081,Y -14.3785,Z 178,A -3.5113,B 6.5238,C 0.2513,E1 6.6877,E2 455.5682} C_DIS
LIN {X 134.5671,Y -10.5238,Z 178,A -1.1477,B 6.5245,C 0.234,E1 6.6882,E2 453.1124} C_DIS
LIN {X 134.9006,Y -4.5718,Z 178,A 0.4911,B 6.5242,C 0.2423,E1 6.6884,E2 451.584} C_DIS
LIN {X 134.9704,Y -1.4526,Z 178,A 1.9384,B 6.5244,C 0.2364,E1 6.6884,E2 450.1202} C_DIS
LIN {X 134.9519,Y 2.5883,Z 178,A 3.8108,B 6.5246,C 0.2288,E1 6.6884,E2 448.2268} C_DIS
LIN {X 134.8445,Y 6.0091,Z 178,A 5.1775,B 6.5247,C 0.2261,E1 6.6882,E2 446.8697} C_DIS
LIN {X 134.5875,Y 10.2453,Z 178,A 6.698,B 6.5247,C 0.2258,E1 6.6879,E2 445.3829} C_DIS
LIN {X 134.2477,Y 14.0107,Z 178,A 8.3082,B 6.5249,C 0.2212,E1 6.6875,E2 443.7708} C_DIS
LIN {X 133.752,Y 18.1474,Z 178,A 9.8903,B 6.5249,C 0.2194,E1 6.6869,E2 442.2107} C_DIS
LIN {X 133.1151,Y 22.3367,Z 178,A 11.731,B 6.5252,C 0.2135,E1 6.6861,E2 440.3634} C_DIS
LIN {X 132.5135,Y 25.6675,Z 178,A 13.1417,B 6.5252,C 0.21,E1 6.6854,E2 438.9549} C_DIS
LIN {X 131.8168,Y 29.0372,Z 178,A 14.7245,B 6.5255,C 0.2038,E1 6.6845,E2 437.3559} C_DIS
LIN {X 130.7941,Y 33.3382,Z 178,A 16.4233,B 6.5255,C 0.2016,E1 6.6834,E2 435.678} C_DIS
LIN {X 129.8355,Y 36.8993,Z 178,A 17.9617,B 6.5257,C 0.1978,E1 6.6822,E2 434.1419} C_DIS
LIN {X 128.7359,Y 40.5689,Z 178,A 19.6891,B 6.5258,C 0.1916,E1 6.6808,E2 432.4009} C_DIS
LIN {X 127.4587,Y 44.4162,Z 178,A 21.2729,B 6.5259,C 0.1893,E1 6.6794,E2 430.8329} C_DIS
LIN {X 125.8268,Y 48.8476,Z 178,A 23.3117,B 6.5261,C 0.1833,E1 6.6773,E2 428.7887} C_DIS
LIN {X 123.8287,Y 53.7116,Z 178,A 25.4212,B 6.5261,C 0.1795,E1 6.6751,E2 426.6931} C_DIS
LIN {X 122.3792,Y 56.9374,Z 178,A 26.9008,B 6.5263,C 0.176,E1 6.6734,E2 425.2154} C_DIS
LIN {X 120.7034,Y 60.4131,Z 178,A 28.5964,B 6.5264,C 0.1709,E1 6.6713,E2 423.5118} C_DIS
LIN {X 118.7758,Y 64.1199,Z 178,A 30.2967,B 6.5264,C 0.1676,E1 6.669,E2 421.8197} C_DIS
LIN {X 116.7363,Y 67.7617,Z 178,A 32.0286,B 6.5266,C 0.1639,E1 6.6667,E2 420.0919} C_DIS
LIN {X 114.5955,Y 71.3222,Z 178,A 33.7655,B 6.5266,C 0.16,E1 6.6641,E2 418.3575} C_DIS
LIN {X 112.3002,Y 74.8843,Z 178,A 35.515,B 6.5268,C 0.1566,E1 6.6614,E2 416.6133} C_DIS
LIN {X 109.8451,Y 78.4413,Z 178,A 37.3405,B 6.5268,C 0.1524,E1 6.6585,E2 414.7882} C_DIS
LIN {X 107.0919,Y 82.1605,Z 178,A 39.6608,B 6.5271,C 0.1421,E1 6.6545,E2 412.4231} C_DIS
LIN {X 104.4133,Y 85.5387,Z 178,A 41.0402,B 6.5271,C 0.1454,E1 6.6522,E2 411.0989} C_DIS
LIN {X 101.5526,Y 88.9162,Z 178,A 42.9211,B 6.5271,C 0.1413,E1 6.6488,E2 409.217} C_DIS
LIN {X 98.5841,Y 92.1968,Z 178,A 45.0796,B 6.5273,C 0.1328,E1 6.6446,E2 407.0236} C_DIS
LIN {X 95.8842,Y 95.0012,Z 178,A 46.2701,B 6.5273,C 0.1369,E1 6.6424,E2 405.8894} C_DIS
LIN {X 93.0916,Y 97.7394,Z 178,A 48.4411,B 6.5274,C 0.1254,E1 6.6379,E2 403.6552} C_DIS
LIN {X 89.8171,Y 100.757,Z 178,A 49.8973,B 6.5274,C 0.1288,E1 6.635,E2 402.2521} C_DIS
LIN {X 86.4873,Y 103.6294,Z 178,A 51.7274,B 6.5274,C 0.1259,E1 6.6311,E2 400.426} C_DIS
LIN {X 83.032,Y 106.4183,Z 178,A 53.6155,B 6.5274,C 0.1225,E1 6.6269,E2 398.5373} C_DIS
LIN {X 79.5283,Y 109.0614,Z 178,A 55.4579,B 6.5275,C 0.1196,E1 6.6228,E2 396.6972} C_DIS
LIN {X 74.7603,Y 112.383,Z 178,A 57.7542,B 6.5275,C 0.1183,E1 6.6176,E2 394.4215} C_DIS
LIN {X 71.5716,Y 114.4403,Z 178,A 59.4849,B 6.5276,C 0.114,E1 6.6134,E2 392.6762} C_DIS
LIN {X 67.6058,Y 116.8266,Z 178,A 61.401,B 6.5276,C 0.1118,E1 6.6088,E2 390.7659} C_DIS
LIN {X 64.0001,Y 118.8402,Z 178,A 63.1492,B 6.5277,C 0.1095,E1 6.6046,E2 389.0183} C_DIS
LIN {X 59.9773,Y 120.9184,Z 178,A 65.0271,B 6.5277,C 0.1077,E1 6.5999,E2 387.1458} C_DIS
LIN {X 56.5356,Y 122.565,Z 178,A 66.5218,B 6.5277,C 0.1076,E1 6.5962,E2 385.6664} C_DIS
LIN {X 53.3061,Y 124.004,Z 178,A 68.0343,B 6.5277,C 0.1057,E1 6.5923,E2 384.1526} C_DIS
LIN {X 49.7381,Y 125.4799,Z 178,A 69.8083,B 6.5278,C 0.1019,E1 6.5876,E2 382.3625} C_DIS
LIN {X 45.2421,Y 127.169,Z 178,A 71.68,B 6.5278,C 0.1023,E1 6.5828,E2 380.5113} C_DIS
LIN {X 41.4105,Y 128.4671,Z 178,A 73.9822,B 6.528,C 0.0921,E1 6.5765,E2 378.1381} C_DIS
LIN {X 36.7383,Y 129.8801,Z 178,A 75.3221,B 6.5279,C 0.1012,E1 6.5731,E2 376.8877} C_DIS
LIN {X 34.3688,Y 130.5276,Z 178,A 76.6195,B 6.5279,C 0.0967,E1 6.5696,E2 375.5598} C_DIS
LIN {X 30.1568,Y 131.564,Z 178,A 78.3218,B 6.5279,C 0.0975,E1 6.565,E2 373.8747} C_DIS
LIN {X 26.5621,Y 132.3371,Z 178,A 79.878,B 6.5279,C 0.0966,E1 6.5607,E2 372.3196} C_DIS
LIN {X 22.5954,Y 133.0719,Z 178,A 81.6543,B 6.5279,C 0.0948,E1 6.5558,E2 370.536} C_DIS
LIN {X 18.7419,Y 133.669,Z 178,A 83.1821,B 6.5279,C 0.0959,E1 6.5516,E2 369.0242} C_DIS
LIN {X 15.1599,Y 134.124,Z 178,A 85.2719,B 6.5281,C 0.0875,E1 6.5457,E2 366.8674} C_DIS
LIN {X 10.714,Y 134.5519,Z 178,A 86.4165,B 6.5279,C 0.0976,E1 6.5427,E2 365.8146} C_DIS
LIN {X 6.0292,Y 134.8436,Z 178,A 88.7738,B 6.5279,C 0.0921,E1 6.536,E2 363.4141} C_DIS
LIN {X 0.3212,Y 134.9766,Z 178,A 91.2995,B 6.528,C 0.0906,E1 6.5289,E2 360.877} C_DIS
LIN {X -4.5853,Y 134.9001,Z 178,A 93.2708,B 6.528,C 0.0922,E1 6.5235,E2 358.9203} C_DIS
LIN {X -8.8704,Y 134.6856,Z 178,A 95.232,B 6.528,C 0.0906,E1 6.518,E2 356.943} C_DIS
LIN {X -13.3612,Y 134.314,Z 178,A 96.9919,B 6.528,C 0.0931,E1 6.5131,E2 355.2026} C_DIS
LIN {X -17.3591,Y 133.8553,Z 178,A 98.6219,B 6.528,C 0.0948,E1 6.5086,E2 353.583} C_DIS
LIN {X -21.2512,Y 133.294,Z 178,A 100.3511,B 6.528,C 0.0947,E1 6.5038,E2 351.8475} C_DIS
LIN {X -25.1816,Y 132.6064,Z 178,A 101.9624,B 6.528,C 0.0966,E1 6.4994,E2 350.247} C_DIS
LIN {X -28.7482,Y 131.8792,Z 178,A 103.4918,B 6.528,C 0.0977,E1 6.4953,E2 348.7206} C_DIS
LIN {X -31.7648,Y 131.1851,Z 178,A 104.8562,B 6.528,C 0.0979,E1 6.4915,E2 347.3508} C_DIS
LIN {X -35.7434,Y 130.1588,Z 178,A 106.8804,B 6.528,C 0.0955,E1 6.486,E2 345.2939} C_DIS
LIN {X -41.0756,Y 128.574,Z 178,A 108.6522,B 6.5278,C 0.105,E1 6.4815,E2 343.5947} C_DIS
LIN {X -44.1117,Y 127.5643,Z 178,A 111.2381,B 6.528,C 0.0905,E1 6.4743,E2 340.8608} C_DIS
LIN {X -50.1566,Y 125.3112,Z 178,A 112.9337,B 6.5278,C 0.1066,E1 6.4702,E2 339.2941} C_DIS
LIN {X -53.8613,Y 123.764,Z 178,A 114.8024,B 6.5278,C 0.1065,E1 6.4653,E2 337.4069} C_DIS
LIN {X -56.9879,Y 122.3559,Z 178,A 116.2648,B 6.5278,C 0.1081,E1 6.4616,E2 335.9447} C_DIS
LIN {X -60.0165,Y 120.899,Z 178,A 117.7634,B 6.5278,C 0.109,E1 6.4578,E2 334.4385} C_DIS
LIN {X -65.4095,Y 118.0703,Z 178,A 120.3882,B 6.5277,C 0.112,E1 6.4514,E2 331.811} C_DIS
LIN {X -67.7691,Y 116.7321,Z 178,A 121.9563,B 6.5277,C 0.1085,E1 6.4475,E2 330.1932} C_DIS
LIN {X -71.2552,Y 114.6372,Z 178,A 123.7504,B 6.5277,C 0.1103,E1 6.4432,E2 328.3923} C_DIS
LIN {X -74.8856,Y 112.2993,Z 178,A 125.0057,B 6.5275,C 0.1202,E1 6.4404,E2 327.2086} C_DIS
LIN {X -77.5243,Y 110.4947,Z 178,A 126.6056,B 6.5275,C 0.1195,E1 6.4367,E2 325.5804} C_DIS
LIN {X -81.2043,Y 107.8187,Z 178,A 128.533,B 6.5275,C 0.1228,E1 6.4324,E2 323.6552} C_DIS
LIN {X -84.6913,Y 105.1017,Z 178,A 130.4222,B 6.5275,C 0.126,E1 6.4282,E2 321.7659} C_DIS
LIN {X -88.1516,Y 102.2168,Z 178,A 132.3814,B 6.5274,C 0.1289,E1 6.424,E2 319.8027} C_DIS
LIN {X -91.6166,Y 99.1238,Z 178,A 134.3797,B 6.5274,C 0.1324,E1 6.4199,E2 317.803} C_DIS
LIN {X -94.837,Y 96.0473,Z 178,A 136.3395,B 6.5272,C 0.1354,E1 6.416,E2 315.8365} C_DIS
LIN {X -98.0312,Y 92.7843,Z 178,A 138.2703,B 6.5272,C 0.1395,E1 6.4122,E2 313.9083} C_DIS
LIN {X -101.0048,Y 89.538,Z 178,A 140.1661,B 6.5271,C 0.1432,E1 6.4087,E2 312.0109} C_DIS
LIN {X -103.7376,Y 86.3575,Z 178,A 142.0056,B 6.5271,C 0.1464,E1 6.4054,E2 310.1657} C_DIS
LIN {X -106.5333,Y 82.8837,Z 178,A 143.9304,B 6.5269,C 0.1503,E1 6.402,E2 308.2388} C_DIS
LIN {X -109.2528,Y 79.2642,Z 178,A 145.8725,B 6.5269,C 0.1545,E1 6.3988,E2 306.296} C_DIS
LIN {X -111.7868,Y 75.6484,Z 178,A 147.9062,B 6.5268,C 0.1571,E1 6.3956,E2 304.2445} C_DIS
LIN {X -115.1054,Y 70.4964,Z 178,A 150.4044,B 6.5266,C 0.1646,E1 6.3919,E2 301.7614} C_DIS
LIN {X -117.3714,Y 66.6559,Z 178,A 152.34,B 6.5265,C 0.1688,E1 6.3891,E2 299.8223} C_DIS
LIN {X -119.2545,Y 63.2225,Z 178,A 154.4534,B 6.5265,C 0.168,E1 6.3863,E2 297.6551} C_DIS
LIN {X -121.1724,Y 59.4624,Z 178,A 155.8166,B 6.5262,C 0.1774,E1 6.3847,E2 296.3461} C_DIS
LIN {X -123.0678,Y 55.4337,Z 178,A 157.5232,B 6.526,C 0.1843,E1 6.3827,E2 294.6635} C_DIS
LIN {X -124.0082,Y 53.2963,Z 178,A 158.7193,B 6.526,C 0.1847,E1 6.3813,E2 293.4434} C_DIS
LIN {X -125.4055,Y 49.9226,Z 178,A 160.2769,B 6.526,C 0.1887,E1 6.3797,E2 291.8864} C_DIS
LIN {X -126.5157,Y 47.0357,Z 178,A 162.0528,B 6.526,C 0.1872,E1 6.3779,E2 290.0549} C_DIS
LIN {X -127.822,Y 43.366,Z 178,A 163.307,B 6.5257,C 0.1961,E1 6.3768,E2 288.8514} C_DIS
LIN {X -128.6854,Y 40.727,Z 178,A 164.5251,B 6.5257,C 0.1988,E1 6.3758,E2 287.6294} C_DIS
LIN {X -129.6445,Y 37.5624,Z 178,A 165.9971,B 6.5255,C 0.202,E1 6.3746,E2 286.1503} C_DIS
LIN {X -130.7185,Y 33.636,Z 178,A 167.7613,B 6.5254,C 0.2064,E1 6.3733,E2 284.3833} C_DIS
LIN {X -131.4767,Y 30.5391,Z 178,A 169.1998,B 6.5254,C 0.2092,E1 6.3724,E2 282.9355} C_DIS
LIN {X -132.2357,Y 27.0604,Z 178,A 170.6593,B 6.5251,C 0.214,E1 6.3716,E2 281.4837} C_DIS
LIN {X -132.8747,Y 23.7244,Z 178,A 172.1458,B 6.5251,C 0.2176,E1 6.3708,E2 279.993} C_DIS
LIN {X -133.4436,Y 20.2852,Z 178,A 173.7761,B 6.5249,C 0.2202,E1 6.3701,E2 278.3455} C_DIS
LIN {X -134.0037,Y 16.1738,Z 178,A 175.4806,B 6.5248,C 0.2258,E1 6.3695,E2 276.6495} C_DIS
LIN {X -134.374,Y 12.7366,Z 178,A 176.9723,B 6.5246,C 0.2297,E1 6.3691,E2 275.156} C_DIS
LIN {X -134.6793,Y 8.9732,Z 178,A 178.6931,B 6.5245,C 0.233,E1 6.3687,E2 273.4221} C_DIS
LIN {X -134.87,Y 5.3553,Z 178,A -179.813,B 6.5243,C 0.2379,E1 6.3685,E2 271.9348} C_DIS
LIN {X -134.9685,Y 1.5907,Z 178,A -178.0774,B 6.5243,C 0.241,E1 6.3685,E2 270.1837} C_DIS
LIN {X -134.9549,Y -2.4101,Z 178,A -176.4317,B 6.524,C 0.2464,E1 6.3685,E2 268.5458} C_DIS
LIN {X -134.8364,Y -6.1724,Z 178,A -174.7228,B 6.5239,C 0.2498,E1 6.3687,E2 266.8246} C_DIS
LIN {X -134.6116,Y -9.9149,Z 178,A -173.1805,B 6.5237,C 0.2548,E1 6.369,E2 265.2895} C_DIS
LIN {X -134.2758,Y -13.7498,Z 178,A -171.3641,B 6.5236,C 0.2575,E1 6.3695,E2 263.4519} C_DIS
LIN {X -133.7844,Y -17.9005,Z 178,A -169.7205,B 6.5233,C 0.264,E1 6.37,E2 261.8257} C_DIS
LIN {X -133.203,Y -21.81,Z 178,A -167.9225,B 6.5232,C 0.2674,E1 6.3708,E2 260.0141} C_DIS
LIN {X -132.5664,Y -25.3905,Z 178,A -166.3893,B 6.523,C 0.2718,E1 6.3716,E2 258.4833} C_DIS
LIN {X -131.9056,Y -28.6259,Z 178,A -164.957,B 6.5229,C 0.2754,E1 6.3724,E2 257.0482} C_DIS
LIN {X -130.2518,Y -35.403,Z 178,A -161.9933,B 6.5225,C 0.2835,E1 6.3744,E2 254.0863} C_DIS
LIN {X -129.1381,Y -39.267,Z 178,A -160.4334,B 6.5222,C 0.2898,E1 6.3756,E2 252.5458} C_DIS
LIN {X -127.8506,Y -43.28,Z 178,A -158.2745,B 6.5222,C 0.2905,E1 6.3776,E2 250.3422} C_DIS
LIN {X -125.9226,Y -48.601,Z 178,A -156.1203,B 6.5218,C 0.2997,E1 6.3796,E2 248.2202} C_DIS
LIN {X -124.3341,Y -52.5338,Z 178,A -154.1057,B 6.5217,C 0.302,E1 6.3818,E2 246.1801} C_DIS
LIN {X -123.1533,Y -55.2425,Z 178,A -152.815,B 6.5215,C 0.3048,E1 6.3832,E2 244.8855} C_DIS
LIN {X -121.6172,Y -58.5479,Z 178,A -151.2173,B 6.5214,C 0.3082,E1 6.3851,E2 243.2824} C_DIS
LIN {X -119.9288,Y -61.9365,Z 178,A -149.0838,B 6.5214,C 0.3062,E1 6.3879,E2 241.0837} C_DIS
LIN {X -117.932,Y -65.6571,Z 178,A -147.3998,B 6.5212,C 0.3119,E1 6.3902,E2 239.4142} C_DIS
LIN {X -116.1311,Y -68.7946,Z 178,A -146.0666,B 6.5209,C 0.318,E1 6.3921,E2 238.1072} C_DIS
LIN {X -113.7773,Y -72.6206,Z 178,A -144.1402,B 6.5207,C 0.3223,E1 6.3949,E2 236.1792} C_DIS
LIN {X -110.1695,Y -77.9854,Z 178,A -141.5147,B 6.5203,C 0.33,E1 6.399,E2 233.5699} C_DIS
LIN {X -105.4546,Y -84.2519,Z 178,A -137.9604,B 6.5201,C 0.3347,E1 6.4051,E2 229.9886} C_DIS
LIN {X -102.5611,Y -87.7519,Z 178,A -136.0042,B 6.5199,C 0.3385,E1 6.4086,E2 228.0294} C_DIS
LIN {X -98.819,Y -91.9445,Z 178,A -133.5688,B 6.5197,C 0.3428,E1 6.4132,E2 225.5885} C_DIS
LIN {X -95.8278,Y -95.058,Z 178,A -131.7199,B 6.5195,C 0.3462,E1 6.4168,E2 223.7381} C_DIS
LIN {X -92.6486,Y -98.1591,Z 178,A -129.8067,B 6.5193,C 0.3495,E1 6.4207,E2 221.8217} C_DIS
LIN {X -89.2894,Y -101.2245,Z 178,A -127.8499,B 6.5191,C 0.3527,E1 6.4247,E2 219.862} C_DIS
LIN {X -85.8224,Y -104.1807,Z 178,A -125.8521,B 6.5191,C 0.3553,E1 6.429,E2 217.8565} C_DIS
LIN {X -82.9247,Y -106.5015,Z 178,A -124.4341,B 6.5188,C 0.3599,E1 6.4321,E2 216.4587} C_DIS
LIN {X -79.3952,Y -109.1576,Z 178,A -122.2625,B 6.5188,C 0.3592,E1 6.4371,E2 214.2498} C_DIS
LIN {X -75.9705,Y -111.5689,Z 178,A -120.5445,B 6.5186,C 0.3627,E1 6.441,E2 212.5396} C_DIS
LIN {X -72.0706,Y -114.1263,Z 178,A -118.5919,B 6.5184,C 0.366,E1 6.4456,E2 210.5905} C_DIS
LIN {X -68.2195,Y -116.4694,Z 178,A -116.6585,B 6.5183,C 0.3683,E1 6.4502,E2 208.6546} C_DIS
LIN {X -64.2731,Y -118.6934,Z 178,A -114.6264,B 6.5183,C 0.3694,E1 6.4552,E2 206.6086} C_DIS
LIN {X -60.839,Y -120.4876,Z 178,A -113.1686,B 6.518,C 0.3738,E1 6.4588,E2 205.1744} C_DIS
LIN {X -57.8688,Y -121.9416,Z 178,A -111.7269,B 6.518,C 0.3749,E1 6.4624,E2 203.7278} C_DIS
LIN {X -54.9052,Y -123.3042,Z 178,A -110.3457,B 6.5178,C 0.3764,E1 6.4659,E2 202.3468} C_DIS
LIN {X -51.6479,Y -124.7041,Z 178,A -108.8153,B 6.5178,C 0.3776,E1 6.4699,E2 200.8132} C_DIS
LIN {X -48.5977,Y -125.9239,Z 178,A -107.3748,B 6.5178,C 0.3783,E1 6.4737,E2 199.3666} C_DIS
LIN {X -44.4489,Y -127.4474,Z 178,A -104.9288,B 6.5181,C 0.3722,E1 6.4803,E2 196.8475} C_DIS
LIN {X -39.8638,Y -128.9552,Z 178,A -103.5633,B 6.5174,C 0.383,E1 6.4837,E2 195.5689} C_DIS
LIN {X -36.2455,Y -130.0183,Z 178,A -101.8617,B 6.5174,C 0.3827,E1 6.4883,E2 193.8541} C_DIS
LIN {X -33.1646,Y -130.8381,Z 178,A -100.4815,B 6.5174,C 0.3832,E1 6.492,E2 192.4701} C_DIS
LIN {X -30.1036,Y -131.5762,Z 178,A -99.158,B 6.5174,C 0.3841,E1 6.4956,E2 191.148} C_DIS
LIN {X -26.7682,Y -132.2952,Z 178,A -97.745,B 6.5174,C 0.3852,E1 6.4995,E2 189.739} C_DIS
LIN {X -23.6264,Y -132.8922,Z 178,A -96.3481,B 6.5174,C 0.3852,E1 6.5033,E2 188.3367} C_DIS
LIN {X -20.0278,Y -133.4834,Z 178,A -94.7265,B 6.5174,C 0.3847,E1 6.5078,E2 186.7052} C_DIS
LIN {X -13.4377,Y -134.3067,Z 178,A -92.0723,B 6.5172,C 0.3877,E1 6.5152,E2 184.0711} C_DIS
LIN {X -10.5006,Y -134.5686,Z 178,A -90.6099,B 6.5173,C 0.3848,E1 6.5193,E2 182.5813} C_DIS
LIN {X -6.8206,Y -134.8038,Z 178,A -88.8817,B 6.5175,C 0.3825,E1 6.5242,E2 180.8316} C_DIS
LIN {X 0.3584,Y -134.9764,Z 178,A -86.1409,B 6.5172,C 0.3868,E1 6.5317,E2 178.1288} C_DIS
LIN {X 0.3584,Y -134.9764,Z 178,A -86.1409,B 6.5172,C 0.3868,E1 6.5317,E2 178.1288} C_DIS
Enddeposition()
LIN {X 0.9869,Y -135.877,Z 178,A -85.7519,B 6.2927,C 0.3879,E1 6.3084,E2 177.8213} C_DIS
Startdeposition()
$VEL.CP = VEL_PRINT
LIN {X -5.0531,Y -135.7867,Z 178,A -88.707,B 6.2923,C 0.3939,E1 6.3,E2 180.8298} C_DIS
LIN {X -10.4986,Y -135.4756,Z 178,A -91.2969,B 6.2921,C 0.3978,E1 6.2927,E2 183.4576} C_DIS
LIN {X -16.3918,Y -134.8884,Z 178,A -93.7752,B 6.2921,C 0.397,E1 6.2858,E2 185.9344} C_DIS
LIN {X -19.98,Y -134.4055,Z 178,A -95.1814,B 6.2922,C 0.395,E1 6.282,E2 187.3259} C_DIS
LIN {X -24.2085,Y -133.7067,Z 178,A -97.0049,B 6.2922,C 0.3945,E1 6.277,E2 189.152} C_DIS
LIN {X -27.3483,Y -133.0999,Z 178,A -98.3665,B 6.2922,C 0.3941,E1 6.2732,E2 190.5157} C_DIS
LIN {X -30.6044,Y -132.3893,Z 178,A -99.7448,B 6.2924,C 0.393,E1 6.2695,E2 191.8909} C_DIS
LIN {X -33.6146,Y -131.6568,Z 178,A -101.1077,B 6.2924,C 0.393,E1 6.2658,E2 193.2614} C_DIS
LIN {X -36.9884,Y -130.7495,Z 178,A -102.6039,B 6.2924,C 0.3924,E1 6.2617,E2 194.7608} C_DIS
LIN {X -43.744,Y -128.6486,Z 178,A -105.5923,B 6.2925,C 0.3902,E1 6.2538,E2 197.7506} C_DIS
LIN {X -46.5508,Y -127.6583,Z 178,A -106.9868,B 6.2925,C 0.3909,E1 6.2501,E2 199.163} C_DIS
LIN {X -50.6507,Y -126.0869,Z 178,A -108.7278,B 6.2927,C 0.3878,E1 6.2456,E2 200.8902} C_DIS
LIN {X -54.0901,Y -124.6501,Z 178,A -110.3158,B 6.2927,C 0.3864,E1 6.2415,E2 202.4805} C_DIS
LIN {X -57.2811,Y -123.2165,Z 178,A -111.7826,B 6.2929,C 0.3847,E1 6.2378,E2 203.9463} C_DIS
LIN {X -60.3757,Y -121.7301,Z 178,A -113.2853,B 6.2929,C 0.3837,E1 6.234,E2 205.4561} C_DIS
LIN {X -64.0731,Y -119.8274,Z 178,A -115.1396,B 6.2929,C 0.3829,E1 6.2293,E2 207.3233} C_DIS
LIN {X -68.0972,Y -117.5869,Z 178,A -117.0473,B 6.2932,C 0.3799,E1 6.2247,E2 209.2266} C_DIS
LIN {X -71.6432,Y -115.4608,Z 178,A -118.8362,B 6.2932,C 0.378,E1 6.2204,E2 211.0213} C_DIS
LIN {X -75.3677,Y -113.0647,Z 178,A -120.7427,B 6.2934,C 0.3757,E1 6.216,E2 212.9325} C_DIS
LIN {X -80.3064,Y -109.6121,Z 178,A -123.0425,B 6.2938,C 0.3689,E1 6.2108,E2 215.2018} C_DIS
LIN {X -82.875,Y -107.6838,Z 178,A -124.6954,B 6.2938,C 0.3702,E1 6.207,E2 216.8922} C_DIS
LIN {X -86.5273,Y -104.771,Z 178,A -126.4143,B 6.2941,C 0.3639,E1 6.2034,E2 218.5792} C_DIS
LIN {X -88.9487,Y -102.7237,Z 178,A -128.0458,B 6.2941,C 0.365,E1 6.1998,E2 220.2476} C_DIS
LIN {X -92.3119,Y -99.7125,Z 178,A -130.0048,B 6.2942,C 0.3621,E1 6.1958,E2 222.2131} C_DIS
LIN {X -95.6504,Y -96.5139,Z 178,A -131.955,B 6.2944,C 0.3583,E1 6.1919,E2 224.1629} C_DIS
LIN {X -98.6872,Y -93.4066,Z 178,A -133.9615,B 6.2945,C 0.3567,E1 6.1879,E2 226.1909} C_DIS
LIN {X -101.7932,Y -90.0113,Z 178,A -135.597,B 6.2949,C 0.3492,E1 6.185,E2 227.7875} C_DIS
LIN {X -104.0552,Y -87.3867,Z 178,A -137.2681,B 6.2949,C 0.3485,E1 6.1819,E2 229.4845} C_DIS
LIN {X -106.8323,Y -83.9689,Z 178,A -139.771,B 6.2948,C 0.3517,E1 6.1774,E2 232.0672} C_DIS
LIN {X -110.0972,Y -79.64,Z 178,A -141.4083,B 6.2955,C 0.3394,E1 6.1749,E2 233.6229} C_DIS
LIN {X -113.5918,Y -74.5711,Z 178,A -144.1405,B 6.2957,C 0.3349,E1 6.1705,E2 236.3711} C_DIS
Enddeposition()
END
